C09002=1025.450,-87.514,-89.281,166.697,46.283,158.451
C09003=1025.445,-87.764,-89.270,166.694,46.286,158.451
C09004=1025.439,-88.014,-89.261,166.691,46.288,158.451
C09005=1025.433,-88.263,-89.250,166.688,46.291,158.451
C09006=1025.427,-88.513,-89.240,166.685,46.294,158.451
C09007=1025.421,-88.763,-89.230,166.683,46.297,158.452
C09008=1025.415,-89.013,-89.221,166.679,46.300,158.452
C09009=1025.409,-89.262,-89.210,166.677,46.302,158.452
C09010=1025.403,-89.512,-89.200,166.673,46.305,158.452
C09011=1025.398,-89.762,-89.190,166.670,46.308,158.452
C09012=1025.392,-90.011,-89.181,166.668,46.311,158.452
C09013=1025.387,-90.262,-89.171,166.664,46.314,158.452
C09014=1025.380,-90.511,-89.160,166.661,46.317,158.452
C09015=1025.375,-90.761,-89.150,166.659,46.319,158.453
C09016=1025.369,-91.011,-89.141,166.655,46.322,158.453
C09017=1025.363,-91.261,-89.130,166.652,46.325,158.453
C09018=1025.358,-91.510,-89.121,166.650,46.328,158.453
C09019=1025.352,-91.760,-89.111,166.646,46.331,158.453
C09020=1025.346,-92.009,-89.101,166.644,46.333,158.453
C09021=1025.340,-92.259,-89.091,166.641,46.336,158.454
C09022=1025.334,-92.509,-89.081,166.637,46.339,158.453
C09023=1025.329,-92.758,-89.071,166.635,46.341,158.454
C09024=1025.323,-93.008,-89.062,166.631,46.345,158.454
C09025=1025.317,-93.258,-89.052,166.628,46.348,158.454
C09026=1025.312,-93.508,-89.042,166.626,46.350,158.454
C09027=1025.305,-93.758,-89.032,166.622,46.353,158.454
C09028=1025.301,-94.007,-89.023,166.620,46.355,158.454
C09029=1025.294,-94.257,-89.013,166.617,46.359,158.455
C09030=1025.289,-94.507,-89.002,166.613,46.361,158.455
C09031=1025.283,-94.756,-88.993,166.611,46.364,158.455
C09032=1025.278,-95.006,-88.983,166.608,46.367,158.455
C09033=1025.272,-95.256,-88.973,166.604,46.369,158.455
C09034=1025.266,-95.506,-88.963,166.602,46.372,158.455
C09035=1025.260,-95.756,-88.954,166.598,46.375,158.455
C09036=1025.255,-96.005,-88.944,166.596,46.378,158.455
C09037=1025.249,-96.255,-88.934,166.593,46.380,158.455
C09038=1025.243,-96.505,-88.924,166.589,46.383,158.456
C09039=1025.238,-96.754,-88.915,166.587,46.386,158.456
C09040=1025.232,-97.004,-88.905,166.584,46.389,158.456
C09041=1025.226,-97.254,-88.895,166.580,46.391,158.456
C09042=1025.220,-97.504,-88.886,166.578,46.394,158.456
C09043=1025.215,-97.753,-88.876,166.575,46.397,158.456
C09044=1025.209,-98.003,-88.867,166.571,46.400,158.456
C09045=1025.203,-98.253,-88.857,166.569,46.403,158.457
C09046=1025.198,-98.502,-88.848,166.566,46.406,158.457
C09047=1025.192,-98.752,-88.838,166.562,46.408,158.457
C09048=1025.186,-99.002,-88.828,166.560,46.411,158.457
C09049=1025.181,-99.251,-88.819,166.557,46.414,158.457
C09050=1025.175,-99.502,-88.810,166.553,46.417,158.457
C09051=1025.168,-99.752,-88.801,166.551,46.420,158.457
C09052=1025.164,-100.001,-88.791,166.548,46.423,158.458
C09053=1025.157,-100.251,-88.781,166.544,46.426,158.458
C09054=1025.152,-100.501,-88.773,166.541,46.429,158.458
C09055=1025.145,-100.786,-88.761,166.538,46.432,158.458
C09056=1025.138,-101.073,-88.750,166.535,46.435,158.458
C09057=1025.132,-101.359,-88.741,166.532,46.439,158.458
C09058=1025.125,-101.644,-88.729,166.527,46.442,158.458
C09059=1025.119,-101.894,-88.720,166.525,46.445,158.459
C09060=1025.113,-102.144,-88.711,166.522,46.448,158.459
C09061=1025.108,-102.394,-88.701,166.518,46.451,158.459
C09062=1025.102,-102.644,-88.692,166.516,46.454,158.459
C09063=1025.097,-102.893,-88.683,166.512,46.456,158.459
C09064=1025.091,-103.143,-88.674,166.509,46.459,158.459
C09065=1025.085,-103.393,-88.665,166.507,46.462,158.460
C09066=1025.079,-103.642,-88.655,166.504,46.465,158.460
C09067=1025.074,-103.892,-88.645,166.500,46.468,158.460
C09068=1025.069,-104.142,-88.637,166.498,46.471,158.460
C09069=1025.062,-104.392,-88.627,166.495,46.474,158.460
C09070=1025.057,-104.641,-88.618,166.491,46.477,158.460
C09071=1025.051,-104.892,-88.609,166.488,46.480,158.460
C09072=1025.045,-105.141,-88.600,166.486,46.482,158.460
C09073=1025.040,-105.391,-88.591,166.482,46.485,158.461
C09074=1025.035,-105.640,-88.581,166.479,46.488,158.461
C09075=1025.029,-105.890,-88.572,166.477,46.491,158.461
C09076=1025.023,-106.141,-88.563,166.473,46.494,158.461
C09077=1025.017,-106.390,-88.554,166.470,46.497,158.461
C09078=1025.011,-106.640,-88.545,166.468,46.500,158.461
C09079=1025.006,-106.889,-88.536,166.465,46.503,158.462
C09080=1025.000,-107.140,-88.527,166.461,46.506,158.462
C09081=1024.994,-107.389,-88.518,166.458,46.509,158.462
C09082=1024.988,-107.639,-88.509,166.455,46.511,158.462
C09083=1024.983,-107.888,-88.500,166.452,46.514,158.462
C09084=1024.977,-108.139,-88.491,166.449,46.517,158.462
C09085=1024.971,-108.388,-88.482,166.447,46.520,158.462
C09086=1024.966,-108.638,-88.473,166.443,46.523,158.462
C09087=1024.960,-108.887,-88.463,166.440,46.526,158.463
C09088=1024.955,-109.137,-88.455,166.437,46.529,158.463
C09089=1024.949,-109.387,-88.446,166.434,46.532,158.463
C09090=1024.943,-109.637,-88.437,166.431,46.535,158.463
C09091=1024.937,-109.887,-88.428,166.428,46.538,158.463
C09092=1024.932,-110.136,-88.419,166.425,46.541,158.463
C09093=1024.926,-110.386,-88.410,166.422,46.544,158.464
C09094=1024.921,-110.636,-88.402,166.419,46.547,158.464
C09095=1024.915,-110.886,-88.392,166.416,46.550,158.464
C09096=1024.909,-111.136,-88.383,166.413,46.553,158.464
C09097=1024.904,-111.385,-88.375,166.410,46.556,158.464
C09098=1024.898,-111.635,-88.365,166.407,46.559,158.464
C09099=1024.893,-111.885,-88.357,166.404,46.562,158.464
C09100=1024.887,-112.135,-88.348,166.401,46.565,158.465
C09101=1024.880,-112.384,-88.339,166.398,46.568,158.465
C09102=1024.875,-112.634,-88.331,166.395,46.571,158.465
C09103=1024.869,-112.884,-88.322,166.391,46.574,158.465
C09104=1024.864,-113.133,-88.313,166.389,46.577,158.465
C09105=1024.858,-113.383,-88.304,166.386,46.580,158.465
C09106=1024.853,-113.633,-88.296,166.383,46.583,158.465
C09107=1024.847,-113.883,-88.287,166.380,46.586,158.466
C09108=1024.841,-114.133,-88.278,166.377,46.589,158.466
C09109=1024.836,-114.383,-88.269,166.374,46.592,158.466
C09110=1024.831,-114.632,-88.261,166.370,46.595,158.466
C09111=1024.825,-114.883,-88.252,166.368,46.598,158.466
C09112=1024.818,-115.132,-88.243,166.365,46.601,158.466
C09113=1024.813,-115.381,-88.235,166.362,46.604,158.467
C09114=1024.807,-115.632,-88.226,166.358,46.607,158.467
C09115=1024.802,-115.881,-88.217,166.356,46.610,158.467
C09116=1024.797,-116.131,-88.209,166.353,46.613,158.467
C09117=1024.791,-116.381,-88.201,166.349,46.616,158.467
C09118=1024.785,-116.631,-88.192,166.346,46.619,158.467
C09119=1024.779,-116.880,-88.183,166.344,46.622,158.467
C09120=1024.774,-117.130,-88.174,166.341,46.625,158.468
C09121=1024.768,-117.379,-88.166,166.337,46.628,158.468
C09122=1024.762,-117.628,-88.157,166.334,46.631,158.468
C09123=1024.757,-117.878,-88.149,166.332,46.634,158.468
C09124=1024.751,-118.127,-88.140,166.328,46.637,158.468
C09125=1024.746,-118.377,-88.132,166.325,46.640,158.468
C09126=1024.740,-118.626,-88.124,166.322,46.643,158.468
C09127=1024.734,-118.876,-88.115,166.320,46.646,158.469
C09128=1024.729,-119.125,-88.107,166.317,46.650,158.469
C09129=1024.724,-119.375,-88.098,166.313,46.653,158.469
///RCONF 1,0,0,0,0,0,0,0,0,0,0,0,0,0,0,0,0,0,0,0,0,0,0,0
C09130=1024.717,-119.625,-88.090,166.310,46.656,158.469
C09131=1024.712,-119.875,-88.082,166.308,46.659,158.469
C09132=1024.707,-120.125,-88.073,166.304,46.662,158.470
C09133=1024.701,-120.374,-88.065,166.301,46.665,158.470
C09134=1024.695,-120.624,-88.057,166.298,46.668,158.470
C09135=1024.690,-120.874,-88.048,166.296,46.671,158.470
C09136=1024.684,-121.124,-88.039,166.292,46.674,158.470
C09137=1024.679,-121.374,-88.031,166.289,46.677,158.470
C09138=1024.673,-121.623,-88.023,166.286,46.680,158.470
C09139=1024.667,-121.909,-88.013,166.283,46.684,158.471
C09140=1024.660,-122.196,-88.004,166.279,46.687,158.471
C09141=1024.654,-122.483,-87.995,166.276,46.691,158.471
C09142=1024.648,-122.769,-87.985,166.272,46.694,158.471
C09143=1024.642,-123.019,-87.977,166.270,46.697,158.471
C09144=1024.636,-123.268,-87.968,166.266,46.700,158.471
C09145=1024.631,-123.518,-87.960,166.263,46.703,158.471
C09146=1024.626,-123.768,-87.951,166.260,46.706,158.472
C09147=1024.619,-124.018,-87.943,166.258,46.709,158.472
C09148=1024.614,-124.268,-87.935,166.254,46.712,158.472
C09149=1024.609,-124.518,-87.927,166.251,46.716,158.472
C09150=1024.603,-124.767,-87.919,166.248,46.719,158.472
C09151=1024.598,-125.017,-87.911,166.246,46.721,158.473
C09152=1024.592,-125.266,-87.903,166.242,46.725,158.473
C09153=1024.587,-125.517,-87.895,166.239,46.728,158.473
C09154=1024.580,-125.767,-87.887,166.236,46.731,158.473
C09155=1024.575,-126.017,-87.878,166.233,46.734,158.473
C09156=1024.570,-126.266,-87.870,166.231,46.737,158.473
C09157=1024.564,-126.516,-87.862,166.227,46.740,158.474
C09158=1024.559,-126.766,-87.854,166.224,46.743,158.474
C09159=1024.553,-127.015,-87.846,166.221,46.747,158.474
C09160=1024.548,-127.265,-87.838,166.218,46.749,158.474
C09161=1024.542,-127.515,-87.830,166.215,46.752,158.474
C09162=1024.537,-127.765,-87.822,166.212,46.756,158.474
C09163=1024.531,-128.014,-87.814,166.209,46.759,158.474
C09164=1024.526,-128.264,-87.805,166.206,46.761,158.475
C09165=1024.522,-128.514,-87.796,166.203,46.764,158.474
C09166=1024.517,-128.763,-87.786,166.200,46.765,158.474
C09167=1024.515,-129.012,-87.776,166.198,46.766,158.474
C09168=1024.511,-129.262,-87.765,166.195,46.767,158.474
C09169=1024.509,-129.512,-87.754,166.193,46.767,158.474
C09170=1024.507,-129.763,-87.741,166.190,46.767,158.473
C09171=1024.506,-130.012,-87.729,166.188,46.766,158.473
C09172=1024.506,-130.262,-87.715,166.186,46.765,158.473
C09173=1024.505,-130.512,-87.702,166.183,46.763,158.472
C09174=1024.505,-130.761,-87.687,166.181,46.760,158.471
C09175=1024.506,-131.011,-87.671,166.179,46.758,158.471
C09176=1024.508,-131.261,-87.657,166.178,46.754,158.470
C09177=1024.510,-131.511,-87.640,166.176,46.751,158.469
C09178=1024.512,-131.760,-87.624,166.175,46.746,158.468
C09179=1024.515,-132.011,-87.606,166.173,46.741,158.467
C09180=1024.519,-132.260,-87.588,166.171,46.736,158.466
C09181=1024.523,-132.510,-87.570,166.169,46.730,158.465
C09182=1024.527,-132.759,-87.551,166.168,46.725,158.464
C09183=1024.230,-132.785,-87.884,166.120,47.002,158.504
C09184=1024.224,-132.536,-87.904,166.122,47.008,158.506
C09185=1024.221,-132.286,-87.923,166.123,47.014,158.507
C09186=1024.217,-132.036,-87.940,166.125,47.019,158.508
C09187=1024.215,-131.786,-87.958,166.126,47.024,158.509
C09188=1024.212,-131.537,-87.975,166.127,47.028,158.510
C09189=1024.209,-131.287,-87.991,166.130,47.032,158.511
C09190=1024.208,-131.037,-88.006,166.131,47.036,158.511
C09191=1024.207,-130.787,-88.022,166.134,47.038,158.512
C09192=1024.207,-130.537,-88.035,166.136,47.040,158.513
C09193=1024.208,-130.287,-88.049,166.137,47.042,158.513
C09194=1024.208,-130.037,-88.062,166.140,47.044,158.514
C09195=1024.209,-129.788,-88.075,166.143,47.044,158.514
C09196=1024.211,-129.539,-88.088,166.145,47.044,158.515
C09197=1024.213,-129.288,-88.100,166.147,47.044,158.515
C09198=1024.216,-129.039,-88.110,166.149,47.044,158.515
C09199=1024.220,-128.789,-88.121,166.152,47.042,158.515
C09200=1024.224,-128.539,-88.130,166.155,47.041,158.515
C09201=1024.228,-128.290,-88.140,166.158,47.039,158.515
C09202=1024.233,-128.040,-88.149,166.161,47.036,158.515
C09203=1024.238,-127.791,-88.156,166.164,47.033,158.515
C09204=1024.243,-127.541,-88.164,166.166,47.030,158.515
C09205=1024.249,-127.292,-88.172,166.170,47.027,158.515
C09206=1024.255,-127.041,-88.181,166.173,47.024,158.515
C09207=1024.260,-126.791,-88.189,166.176,47.020,158.514
C09208=1024.266,-126.541,-88.196,166.180,47.017,158.514
C09209=1024.271,-126.292,-88.205,166.182,47.014,158.514
C09210=1024.277,-126.042,-88.213,166.185,47.011,158.514
C09211=1024.282,-125.792,-88.221,166.188,47.008,158.514
C09212=1024.288,-125.543,-88.228,166.191,47.004,158.514
C09213=1024.294,-125.293,-88.237,166.195,47.001,158.514
C09214=1024.299,-125.043,-88.244,166.198,46.998,158.513
C09215=1024.305,-124.793,-88.253,166.200,46.995,158.513
C09216=1024.310,-124.543,-88.261,166.203,46.992,158.513
C09217=1024.316,-124.293,-88.269,166.206,46.988,158.513
C09218=1024.322,-124.044,-88.278,166.210,46.985,158.513
C09219=1024.327,-123.793,-88.286,166.213,46.982,158.513
C09220=1024.333,-123.544,-88.293,166.215,46.979,158.512
C09221=1024.338,-123.294,-88.302,166.218,46.976,158.512
C09222=1024.343,-123.044,-88.310,166.221,46.973,158.512
C09223=1024.349,-122.795,-88.318,166.225,46.969,158.512
C09224=1024.354,-122.545,-88.327,166.228,46.966,158.512
C09225=1024.360,-122.295,-88.336,166.230,46.963,158.512
C09226=1024.366,-122.045,-88.343,166.233,46.960,158.511
C09227=1024.371,-121.795,-88.351,166.237,46.957,158.511
C09228=1024.376,-121.545,-88.360,166.240,46.954,158.511
C09229=1024.382,-121.296,-88.368,166.242,46.951,158.511
C09230=1024.388,-121.046,-88.376,166.245,46.948,158.511
C09231=1024.394,-120.796,-88.385,166.249,46.944,158.511
C09232=1024.399,-120.546,-88.394,166.252,46.941,158.510
C09233=1024.405,-120.297,-88.401,166.255,46.938,158.510
C09234=1024.410,-120.047,-88.410,166.257,46.935,158.510
C09235=1024.415,-119.797,-88.418,166.261,46.932,158.510
C09236=1024.421,-119.547,-88.427,166.264,46.929,158.510
C09237=1024.427,-119.298,-88.435,166.267,46.926,158.510
C09238=1024.433,-119.048,-88.444,166.270,46.922,158.510
C09239=1024.438,-118.798,-88.452,166.272,46.920,158.509
C09240=1024.444,-118.548,-88.461,166.276,46.916,158.509
C09241=1024.450,-118.298,-88.469,166.279,46.913,158.509
C09242=1024.455,-118.049,-88.477,166.282,46.910,158.509
C09243=1024.460,-117.799,-88.486,166.286,46.907,158.509
C09244=1024.467,-117.513,-88.496,166.289,46.903,158.509
C09245=1024.473,-117.228,-88.505,166.292,46.900,158.508
C09246=1024.480,-116.942,-88.514,166.296,46.896,158.508
C09247=1024.486,-116.656,-88.525,166.299,46.893,158.508
C09248=1024.491,-116.407,-88.533,166.302,46.890,158.508
C09249=1024.497,-116.157,-88.541,166.305,46.887,158.508
C09250=1024.503,-115.907,-88.551,166.308,46.883,158.508
C09251=1024.509,-115.658,-88.559,166.311,46.880,158.507
C09252=1024.514,-115.408,-88.568,166.314,46.877,158.507
C09253=1024.520,-115.158,-88.577,166.317,46.874,158.507
C09254=1024.526,-114.908,-88.585,166.320,46.871,158.507
C09255=1024.531,-114.658,-88.593,166.323,46.868,158.507
C09256=1024.536,-114.409,-88.602,166.326,46.865,158.507
C09257=1024.543,-114.159,-88.611,166.330,46.862,158.507
C09258=1024.548,-113.909,-88.620,166.332,46.859,158.506
C09259=1024.554,-113.659,-88.628,166.335,46.856,158.506
C09260=1024.559,-113.409,-88.637,166.338,46.853,158.506
C09261=1024.564,-113.160,-88.646,166.342,46.850,158.506
C09262=1024.570,-112.910,-88.655,166.344,46.847,158.506
C09263=1024.576,-112.660,-88.664,166.347,46.844,158.506
C09264=1024.582,-112.410,-88.671,166.350,46.841,158.506
C09265=1024.588,-112.161,-88.681,166.354,46.838,158.505
C09266=1024.593,-111.911,-88.689,166.357,46.835,158.505
C09267=1024.598,-111.661,-88.698,166.359,46.832,158.505
C09268=1024.604,-111.411,-88.708,166.363,46.829,158.505
C09269=1024.610,-111.162,-88.716,166.366,46.825,158.505
C09270=1024.616,-110.911,-88.725,166.369,46.822,158.505
C09271=1024.621,-110.662,-88.734,166.371,46.819,158.504
C09272=1024.626,-110.412,-88.743,166.374,46.816,158.504
C09273=1024.632,-110.162,-88.751,166.378,46.813,158.504
C09274=1024.638,-109.913,-88.761,166.381,46.810,158.504
C09275=1024.644,-109.663,-88.769,166.383,46.807,158.504
C09276=1024.649,-109.413,-88.778,166.386,46.804,158.504
C09277=1024.655,-109.163,-88.787,166.390,46.801,158.503
C09278=1024.660,-108.913,-88.796,166.393,46.798,158.503
C09279=1024.666,-108.664,-88.805,166.396,46.795,158.503
C09280=1024.672,-108.420,-88.814,166.399,46.792,158.503
C09281=1024.678,-108.177,-88.822,166.402,46.789,158.503
C09282=1024.683,-107.935,-88.831,166.405,46.786,158.503
C09283=1024.689,-107.691,-88.840,166.407,46.783,158.503
C09284=1024.694,-107.447,-88.848,166.411,46.780,158.502
C09285=1024.700,-107.204,-88.858,166.414,46.777,158.502
C09286=1024.705,-106.961,-88.866,166.416,46.774,158.502
C09287=1024.711,-106.717,-88.875,166.420,46.772,158.502
C09288=1024.716,-106.468,-88.884,166.423,46.769,158.502
C09289=1024.722,-106.218,-88.893,166.425,46.766,158.502
C09290=1024.728,-105.969,-88.902,166.429,46.763,158.502
C09291=1024.733,-105.718,-88.911,166.432,46.760,158.502
C09292=1024.738,-105.469,-88.921,166.435,46.757,158.501
C09293=1024.745,-105.219,-88.930,166.437,46.754,158.501
C09294=1024.750,-104.969,-88.939,166.441,46.751,158.501
C09295=1024.756,-104.720,-88.948,166.444,46.748,158.501
C09296=1024.761,-104.470,-88.957,166.446,46.745,158.501
C09297=1024.768,-104.220,-88.966,166.449,46.742,158.501
C09298=1024.773,-103.970,-88.977,166.453,46.739,158.500
C09299=1024.778,-103.720,-88.985,166.456,46.735,158.500
C09300=1024.784,-103.470,-88.995,166.458,46.733,158.500
C09301=1024.790,-103.221,-89.003,166.462,46.730,158.500
C09302=1024.796,-102.971,-89.013,166.465,46.727,158.500
C09303=1024.801,-102.722,-89.022,166.468,46.723,158.500
C09304=1024.807,-102.471,-89.031,166.470,46.721,158.500
C09305=1024.813,-102.221,-89.041,166.474,46.718,158.499
C09306=1024.818,-101.972,-89.050,166.477,46.714,158.499
C09307=1024.824,-101.722,-89.059,166.480,46.711,158.499
C09308=1024.831,-101.423,-89.070,166.483,46.708,158.499
C09309=1024.838,-101.125,-89.082,166.486,46.705,158.499
C09310=1024.844,-100.826,-89.092,166.491,46.701,158.499
C09311=1024.851,-100.527,-89.104,166.494,46.698,158.498
C09312=1024.857,-100.277,-89.114,166.497,46.694,158.498
C09313=1024.863,-100.027,-89.122,166.500,46.691,158.498
C09314=1024.869,-99.778,-89.132,166.504,46.688,158.498
C09315=1024.874,-99.528,-89.142,166.506,46.686,158.498
C09316=1024.880,-99.278,-89.151,166.509,46.682,158.498
C09317=1024.886,-99.028,-89.160,166.512,46.679,158.498
C09318=1024.892,-98.779,-89.169,166.516,46.676,158.497
C09319=1024.898,-98.529,-89.179,166.518,46.673,158.497
C09320=1024.904,-98.280,-89.188,166.521,46.670,158.497
C09321=1024.909,-98.030,-89.198,166.525,46.667,158.497
C09322=1024.915,-97.779,-89.207,166.528,46.664,158.497
C09323=1024.920,-97.530,-89.216,166.530,46.662,158.497
C09324=1024.926,-97.280,-89.227,166.534,46.659,158.497
C09325=1024.932,-97.030,-89.236,166.537,46.656,158.496
C09326=1024.937,-96.781,-89.246,166.539,46.653,158.496
C09327=1024.943,-96.531,-89.255,166.543,46.650,158.496
C09328=1024.949,-96.281,-89.266,166.546,46.648,158.496
C09329=1024.954,-96.032,-89.275,166.548,46.645,158.496
C09330=1024.960,-95.782,-89.284,166.552,46.642,158.496
C09331=1024.966,-95.532,-89.295,166.555,46.639,158.496
C09332=1024.972,-95.282,-89.304,166.557,46.636,158.495
C09333=1024.977,-95.033,-89.314,166.561,46.634,158.495
C09334=1024.983,-94.783,-89.323,166.564,46.631,158.495
C09335=1024.988,-94.533,-89.334,166.566,46.628,158.495
C09336=1024.994,-94.283,-89.343,166.570,46.625,158.495
C09337=1024.999,-94.033,-89.353,166.573,46.622,158.495
C09338=1025.005,-93.784,-89.363,166.575,46.619,158.495
C09339=1025.011,-93.534,-89.373,166.579,46.617,158.495
C09340=1025.017,-93.284,-89.382,166.582,46.613,158.494
C09341=1025.022,-93.035,-89.393,166.584,46.611,158.494
C09342=1025.028,-92.785,-89.402,166.587,46.608,158.494
C09343=1025.034,-92.535,-89.413,166.591,46.605,158.494
C09344=1025.040,-92.285,-89.422,166.593,46.602,158.494
C09345=1025.046,-92.036,-89.431,166.597,46.599,158.494
C09346=1025.051,-91.786,-89.441,166.600,46.596,158.494
C09347=1025.057,-91.536,-89.451,166.602,46.594,158.493
C09348=1025.063,-91.286,-89.461,166.605,46.590,158.493
C09349=1025.069,-91.036,-89.471,166.609,46.587,158.493
C09350=1025.075,-90.787,-89.482,166.611,46.585,158.493
C09351=1025.080,-90.538,-89.491,166.615,46.582,158.493
C09352=1025.086,-90.288,-89.501,166.618,46.579,158.493
C09353=1025.092,-90.038,-89.511,166.620,46.576,158.493
C09354=1025.097,-89.788,-89.521,166.623,46.573,158.492
C09355=1025.104,-89.539,-89.531,166.627,46.570,158.492
C09356=1025.109,-89.288,-89.541,166.629,46.567,158.492
C09357=1025.115,-89.039,-89.550,166.632,46.565,158.492
C09358=1025.120,-88.789,-89.561,166.636,46.562,158.492
C09359=1025.126,-88.539,-89.570,166.638,46.559,158.492
C09360=1025.132,-88.290,-89.581,166.641,46.556,158.492
C09361=1025.138,-88.040,-89.591,166.645,46.553,158.491
C09362=1025.144,-87.790,-89.601,166.647,46.550,158.491
C09363=1025.150,-87.540,-89.610,166.650,46.547,158.491
C09364=1025.155,-87.291,-89.621,166.654,46.545,158.491
C09365=1025.162,-87.041,-89.631,166.657,46.542,158.491
C09366=1025.167,-86.791,-89.641,166.659,46.539,158.491
C09367=1025.173,-86.542,-89.651,166.663,46.536,158.491
C09368=1025.178,-86.292,-89.661,166.666,46.533,158.491
C09369=1025.185,-86.042,-89.671,166.668,46.530,158.490
C09370=1025.190,-85.792,-89.681,166.671,46.527,158.490
C09371=1025.196,-85.543,-89.692,166.675,46.525,158.490
C09372=1025.203,-85.259,-89.703,166.678,46.521,158.490
C09373=1025.210,-84.975,-89.714,166.681,46.518,158.490
C09374=1025.216,-84.691,-89.725,166.685,46.515,158.490
C09375=1025.223,-84.408,-89.737,166.688,46.511,158.489
C09376=1025.229,-84.158,-89.747,166.691,46.509,158.489
C09377=1025.235,-83.908,-89.758,166.694,46.506,158.489
C09378=1025.241,-83.659,-89.768,166.697,46.503,158.489
C09379=1025.246,-83.409,-89.778,166.700,46.500,158.489
C09380=1025.253,-83.159,-89.788,166.703,46.497,158.489
C09381=1025.258,-82.909,-89.798,166.707,46.494,158.489
C09382=1025.265,-82.660,-89.809,166.709,46.491,158.488
C09383=1025.270,-82.410,-89.819,166.712,46.488,158.488
C09384=1025.276,-82.160,-89.828,166.715,46.485,158.488
C09385=1025.282,-81.911,-89.839,166.718,46.482,158.488
C09386=1025.288,-81.661,-89.849,166.721,46.480,158.488
C09387=1025.294,-81.411,-89.860,166.724,46.477,158.488
C09388=1025.300,-81.162,-89.869,166.727,46.474,158.487
C09389=1025.306,-80.912,-89.880,166.730,46.471,158.487
C09390=1025.311,-80.662,-89.890,166.733,46.468,158.487
C09391=1025.318,-80.413,-89.901,166.736,46.465,158.487
C09392=1025.323,-80.163,-89.911,166.739,46.462,158.487
C09393=1025.330,-79.913,-89.921,166.742,46.459,158.487
C09394=1025.336,-79.663,-89.932,166.744,46.456,158.486
C09395=1025.341,-79.413,-89.942,166.748,46.454,158.486
C09396=1025.347,-79.164,-89.953,166.751,46.451,158.486
C09397=1025.352,-78.914,-89.963,166.754,46.448,158.486
C09398=1025.359,-78.664,-89.974,166.757,46.446,158.486
C09399=1025.365,-78.415,-89.985,166.759,46.443,158.486
C09400=1025.370,-78.165,-89.995,166.763,46.440,158.486
C09401=1025.376,-77.915,-90.006,166.766,46.437,158.486
C09402=1025.382,-77.666,-90.017,166.768,46.435,158.486
C09403=1025.388,-77.416,-90.026,166.772,46.432,158.485
C09404=1025.394,-77.166,-90.037,166.775,46.429,158.485
C09405=1025.400,-76.916,-90.048,166.777,46.426,158.485
C09406=1025.405,-76.666,-90.058,166.781,46.424,158.485
C09407=1025.411,-76.417,-90.069,166.783,46.421,158.485
C09408=1025.417,-76.167,-90.080,166.786,46.418,158.485
C09409=1025.423,-75.918,-90.090,166.790,46.415,158.484
C09410=1025.429,-75.668,-90.101,166.792,46.412,158.484
C09411=1025.435,-75.418,-90.112,166.796,46.410,158.484
C09412=1025.441,-75.168,-90.123,166.798,46.407,158.484
C09413=1025.446,-74.919,-90.134,166.801,46.404,158.484
C09414=1025.453,-74.669,-90.143,166.804,46.401,158.484
C09415=1025.458,-74.420,-90.154,166.807,46.399,158.484
C09416=1025.464,-74.170,-90.165,166.810,46.396,158.484
C09417=1025.470,-73.920,-90.176,166.813,46.393,158.483
C09418=1025.476,-73.670,-90.187,166.816,46.390,158.483
C09419=1025.481,-73.421,-90.198,166.818,46.388,158.483
C09420=1025.487,-73.170,-90.209,166.822,46.385,158.483
C09421=1025.492,-72.921,-90.220,166.825,46.382,158.483
C09422=1025.499,-72.671,-90.231,166.827,46.380,158.483
C09423=1025.504,-72.421,-90.242,166.831,46.377,158.483
C09424=1025.510,-72.172,-90.253,166.833,46.374,158.483
C09425=1025.516,-71.922,-90.263,166.837,46.372,158.483
C09426=1025.522,-71.673,-90.274,166.839,46.369,158.482
C09427=1025.528,-71.423,-90.286,166.842,46.366,158.482
C09428=1025.533,-71.173,-90.297,166.845,46.364,158.482
C09429=1025.539,-70.923,-90.308,166.848,46.361,158.482
C09430=1025.544,-70.674,-90.319,166.851,46.359,158.482
C09431=1025.550,-70.424,-90.330,166.854,46.356,158.482
C09432=1025.557,-70.174,-90.341,166.856,46.353,158.481
C09433=1025.562,-69.925,-90.352,166.860,46.351,158.481
C09434=1025.568,-69.675,-90.363,166.863,46.348,158.481
C09435=1025.574,-69.426,-90.374,166.866,46.346,158.481
C09436=1025.580,-69.144,-90.387,166.869,46.343,158.481
C09437=1025.587,-68.863,-90.399,166.872,46.340,158.481
C09438=1025.593,-68.581,-90.412,166.876,46.337,158.481
C09439=1025.600,-68.299,-90.424,166.879,46.334,158.481
C09440=1025.605,-68.050,-90.436,166.882,46.331,158.481
C09441=1025.612,-67.800,-90.447,166.885,46.329,158.480
C09442=1025.618,-67.550,-90.458,166.888,46.326,158.480
C09443=1025.623,-67.301,-90.469,166.890,46.323,158.480
C09444=1025.630,-67.051,-90.480,166.894,46.320,158.480
C09445=1025.635,-66.801,-90.491,166.896,46.318,158.480
C09446=1025.641,-66.552,-90.502,166.899,46.315,158.480
C09447=1025.647,-66.301,-90.514,166.902,46.313,158.480
///RCONF 1,0,0,1,0,0,0,0,0,0,0,0,0,0,0,0,0,0,0,0,0,0,0,0
C09448=1025.653,-66.052,-90.525,166.905,46.310,158.479
C09449=1025.658,-65.803,-90.536,166.908,46.307,158.479
C09450=1025.665,-65.553,-90.547,166.911,46.304,158.479
C09451=1025.671,-65.303,-90.558,166.914,46.301,158.479
C09452=1025.676,-65.054,-90.569,166.917,46.299,158.479
C09453=1025.683,-64.803,-90.580,166.920,46.296,158.479
C09454=1025.688,-64.554,-90.592,166.923,46.294,158.479
C09455=1025.694,-64.304,-90.604,166.926,46.291,158.479
C09456=1025.700,-64.054,-90.615,166.928,46.288,158.478
C09457=1025.706,-63.805,-90.625,166.932,46.285,158.478
C09458=1025.712,-63.555,-90.637,166.934,46.283,158.478
C09459=1025.718,-63.306,-90.648,166.937,46.280,158.478
C09460=1025.723,-63.056,-90.660,166.940,46.278,158.478
C09461=1025.729,-62.806,-90.671,166.943,46.275,158.478
C09462=1025.736,-62.557,-90.683,166.946,46.272,158.478
C09463=1025.742,-62.307,-90.694,166.949,46.269,158.477
C09464=1025.748,-62.057,-90.705,166.952,46.266,158.477
C09465=1025.754,-61.807,-90.716,166.955,46.264,158.477
C09466=1025.759,-61.558,-90.728,166.958,46.261,158.477
C09467=1025.765,-61.309,-90.739,166.960,46.258,158.477
C09468=1025.771,-61.058,-90.750,166.964,46.256,158.477
C09469=1025.777,-60.809,-90.762,166.966,46.253,158.477
C09470=1025.784,-60.559,-90.773,166.969,46.250,158.476
C09471=1025.789,-60.310,-90.784,166.972,46.248,158.476
C09472=1025.795,-60.060,-90.797,166.975,46.245,158.476
C09473=1025.801,-59.810,-90.807,166.978,46.243,158.476
C09474=1025.807,-59.560,-90.819,166.981,46.240,158.476
C09475=1025.814,-59.311,-90.830,166.984,46.237,158.476
C09476=1025.820,-59.061,-90.842,166.987,46.234,158.476
C09477=1025.825,-58.812,-90.854,166.990,46.231,158.475
C09478=1025.831,-58.562,-90.865,166.992,46.229,158.475
C09479=1025.837,-58.312,-90.876,166.996,46.226,158.475
C09480=1025.844,-58.063,-90.888,166.998,46.224,158.475
C09481=1025.850,-57.813,-90.899,167.002,46.221,158.475
C09482=1025.856,-57.563,-90.911,167.004,46.218,158.475
C09483=1025.861,-57.314,-90.922,167.007,46.215,158.475
C09484=1025.868,-57.064,-90.934,167.009,46.213,158.474
C09485=1025.874,-56.814,-90.945,167.013,46.210,158.474
C09486=1025.880,-56.565,-90.956,167.016,46.207,158.474
C09487=1025.886,-56.315,-90.969,167.019,46.205,158.474
C09488=1025.892,-56.065,-90.980,167.022,46.202,158.474
C09489=1025.898,-55.816,-90.992,167.024,46.199,158.474
C09490=1025.904,-55.566,-91.002,167.028,46.196,158.474
C09491=1025.911,-55.317,-91.014,167.030,46.194,158.473
C09492=1025.916,-55.066,-91.026,167.033,46.191,158.473
C09493=1025.922,-54.817,-91.038,167.036,46.189,158.473
C09494=1025.929,-54.567,-91.049,167.039,46.186,158.473
C09495=1025.935,-54.318,-91.061,167.041,46.183,158.473
C09496=1025.941,-54.069,-91.073,167.045,46.180,158.473
C09497=1025.947,-53.818,-91.084,167.047,46.178,158.472
C09498=1025.953,-53.569,-91.096,167.051,46.175,158.472
C09499=1025.959,-53.319,-91.107,167.054,46.172,158.472
C09500=1025.966,-53.039,-91.120,167.057,46.169,158.472
C09501=1025.973,-52.758,-91.134,167.060,46.166,158.472
C09502=1025.980,-52.478,-91.147,167.064,46.163,158.472
C09503=1025.987,-52.197,-91.160,167.066,46.160,158.471
C09504=1025.993,-51.948,-91.172,167.069,46.157,158.471
C09505=1025.999,-51.699,-91.183,167.073,46.154,158.471
C09506=1026.005,-51.448,-91.195,167.075,46.151,158.471
C09507=1026.012,-51.199,-91.207,167.078,46.148,158.471
C09508=1026.018,-50.950,-91.219,167.081,46.146,158.471
C09509=1026.024,-50.700,-91.230,167.084,46.143,158.471
C09510=1026.030,-50.450,-91.242,167.086,46.140,158.470
C09511=1026.035,-50.201,-91.255,167.090,46.138,158.470
C09512=1026.042,-49.951,-91.266,167.092,46.135,158.470
C09513=1026.048,-49.701,-91.278,167.095,46.133,158.470
C09514=1026.053,-49.451,-91.291,167.098,46.130,158.470
C09515=1026.060,-49.202,-91.302,167.101,46.128,158.470
C09516=1026.065,-48.952,-91.315,167.104,46.125,158.470
C09517=1026.071,-48.703,-91.327,167.106,46.123,158.469
C09518=1026.077,-48.453,-91.339,167.110,46.120,158.469
C09519=1026.083,-48.203,-91.351,167.112,46.118,158.469
C09520=1026.090,-47.953,-91.363,167.114,46.115,158.469
C09521=1026.095,-47.704,-91.375,167.118,46.112,158.469
C09522=1026.102,-47.454,-91.387,167.120,46.110,158.469
C09523=1026.108,-47.204,-91.400,167.124,46.107,158.469
C09524=1026.113,-46.955,-91.412,167.126,46.105,158.469
C09525=1026.119,-46.706,-91.424,167.129,46.102,158.468
C09526=1026.125,-46.456,-91.436,167.132,46.100,158.468
C09527=1026.131,-46.206,-91.449,167.135,46.097,158.468
C09528=1026.137,-45.956,-91.460,167.138,46.094,158.468
C09529=1026.143,-45.707,-91.472,167.140,46.092,158.468
C09530=1026.150,-45.457,-91.484,167.143,46.089,158.468
C09531=1026.155,-45.207,-91.497,167.146,46.087,158.468
C09532=1026.161,-44.958,-91.509,167.149,46.084,158.467
C09533=1026.167,-44.708,-91.521,167.152,46.082,158.467
C09534=1026.173,-44.458,-91.534,167.155,46.079,158.467
C09535=1026.179,-44.209,-91.546,167.157,46.076,158.467
C09536=1026.185,-43.960,-91.558,167.160,46.074,158.467
C09537=1026.191,-43.710,-91.570,167.163,46.071,158.467
C09538=1026.198,-43.460,-91.582,167.166,46.069,158.467
C09539=1026.204,-43.210,-91.595,167.169,46.066,158.466
C09540=1026.210,-42.961,-91.607,167.171,46.063,158.466
C09541=1026.216,-42.712,-91.619,167.175,46.061,158.466
C09542=1026.222,-42.462,-91.631,167.177,46.058,158.466
C09543=1026.228,-42.212,-91.644,167.180,46.056,158.466
C09544=1026.234,-41.962,-91.656,167.183,46.053,158.466
C09545=1026.240,-41.713,-91.669,167.185,46.050,158.465
C09546=1026.246,-41.463,-91.682,167.189,46.048,158.465
C09547=1026.253,-41.214,-91.694,167.191,46.045,158.465
C09548=1026.258,-40.964,-91.706,167.194,46.042,158.465
C09549=1026.264,-40.715,-91.719,167.197,46.040,158.465
C09550=1026.271,-40.465,-91.730,167.200,46.037,158.465
C09551=1026.277,-40.215,-91.743,167.203,46.035,158.465
C09552=1026.283,-39.965,-91.755,167.205,46.033,158.464
C09553=1026.289,-39.716,-91.768,167.208,46.030,158.464
C09554=1026.295,-39.466,-91.780,167.211,46.028,158.464
C09555=1026.302,-39.217,-91.793,167.214,46.025,158.464
C09556=1026.307,-38.968,-91.805,167.217,46.022,158.464
C09557=1026.313,-38.718,-91.818,167.219,46.020,158.464
C09558=1026.319,-38.468,-91.830,167.222,46.017,158.464
C09559=1026.325,-38.218,-91.843,167.225,46.015,158.463
C09560=1026.331,-37.969,-91.856,167.228,46.012,158.463
C09561=1026.337,-37.719,-91.868,167.231,46.010,158.463
C09562=1026.343,-37.469,-91.881,167.233,46.007,158.463
C09563=1026.349,-37.220,-91.894,167.237,46.005,158.463
C09564=1026.356,-36.940,-91.907,167.239,46.002,158.463
C09565=1026.363,-36.660,-91.922,167.242,45.999,158.463
C09566=1026.370,-36.380,-91.936,167.246,45.997,158.463
C09567=1026.377,-36.100,-91.951,167.249,45.994,158.462
C09568=1026.382,-35.850,-91.963,167.251,45.991,158.462
C09569=1026.389,-35.601,-91.976,167.254,45.989,158.462
C09570=1026.395,-35.351,-91.989,167.257,45.986,158.462
C09571=1026.401,-35.101,-92.002,167.260,45.984,158.462
C09572=1026.407,-34.852,-92.015,167.262,45.981,158.462
C09573=1026.413,-34.602,-92.027,167.266,45.979,158.462
C09574=1026.418,-34.353,-92.040,167.268,45.976,158.461
C09575=1026.424,-34.103,-92.053,167.271,45.974,158.461
C09576=1026.431,-33.854,-92.065,167.274,45.971,158.461
C09577=1026.437,-33.604,-92.078,167.276,45.968,158.461
C09578=1026.443,-33.355,-92.091,167.280,45.966,158.461
C09579=1026.449,-33.105,-92.103,167.282,45.963,158.461
C09580=1026.455,-32.855,-92.116,167.284,45.961,158.460
C09581=1026.461,-32.606,-92.129,167.288,45.958,158.460
C09582=1026.467,-32.356,-92.142,167.290,45.956,158.460
C09583=1026.473,-32.106,-92.155,167.293,45.953,158.460
C09584=1026.479,-31.857,-92.168,167.296,45.951,158.460
C09585=1026.485,-31.607,-92.181,167.298,45.948,158.460
C09586=1026.491,-31.358,-92.194,167.302,45.946,158.460
C09587=1026.498,-31.107,-92.207,167.304,45.943,158.459
C09588=1026.504,-30.858,-92.220,167.307,45.940,158.459
C09589=1026.510,-30.608,-92.233,167.310,45.938,158.459
C09590=1026.516,-30.359,-92.246,167.312,45.935,158.459
C09591=1026.522,-30.109,-92.258,167.315,45.933,158.459
C09592=1026.529,-29.860,-92.271,167.318,45.930,158.459
C09593=1026.535,-29.610,-92.284,167.321,45.928,158.458
C09594=1026.541,-29.361,-92.297,167.323,45.926,158.458
C09595=1026.547,-29.111,-92.310,167.326,45.923,158.458
C09596=1026.553,-28.862,-92.323,167.329,45.920,158.458
C09597=1026.559,-28.612,-92.335,167.332,45.918,158.458
C09598=1026.566,-28.363,-92.349,167.335,45.915,158.458
C09599=1026.571,-28.113,-92.361,167.337,45.913,158.458
C09600=1026.578,-27.864,-92.374,167.340,45.910,158.457
C09601=1026.584,-27.614,-92.388,167.343,45.908,158.457
C09602=1026.590,-27.364,-92.401,167.345,45.905,158.457
C09603=1026.597,-27.114,-92.414,167.349,45.903,158.457
C09604=1026.603,-26.865,-92.427,167.351,45.900,158.457
C09605=1026.608,-26.615,-92.440,167.354,45.898,158.457
C09606=1026.614,-26.366,-92.454,167.356,45.895,158.457
C09607=1026.620,-26.116,-92.467,167.359,45.893,158.457
C09608=1026.626,-25.867,-92.479,167.362,45.890,158.456
C09609=1026.632,-25.617,-92.493,167.364,45.888,158.456
C09610=1026.639,-25.367,-92.507,167.368,45.886,158.456
C09611=1026.645,-25.118,-92.520,167.370,45.883,158.456
C09612=1026.651,-24.868,-92.533,167.373,45.881,158.456
C09613=1026.657,-24.619,-92.546,167.375,45.878,158.456
C09614=1026.662,-24.369,-92.560,167.379,45.876,158.456
C09615=1026.669,-24.120,-92.573,167.381,45.873,158.455
C09616=1026.675,-23.871,-92.586,167.383,45.871,158.455
C09617=1026.681,-23.620,-92.599,167.387,45.868,158.455
C09618=1026.687,-23.370,-92.613,167.389,45.866,158.455
C09619=1026.693,-23.121,-92.626,167.391,45.863,158.455
C09620=1026.699,-22.872,-92.640,167.394,45.861,158.455
C09621=1026.705,-22.623,-92.653,167.397,45.858,158.454
C09622=1026.711,-22.372,-92.666,167.400,45.856,158.454
C09623=1026.717,-22.122,-92.680,167.402,45.854,158.454
C09624=1026.724,-21.873,-92.693,167.406,45.851,158.454
C09625=1026.730,-21.624,-92.706,167.408,45.849,158.454
C09626=1026.736,-21.375,-92.720,167.411,45.846,158.454
C09627=1026.742,-21.125,-92.733,167.413,45.844,158.454
C09628=1026.749,-20.844,-92.748,167.416,45.841,158.453
C09629=1026.756,-20.563,-92.764,167.420,45.839,158.453
C09630=1026.763,-20.282,-92.778,167.423,45.836,158.453
C09631=1026.770,-20.001,-92.794,167.425,45.833,158.453
C09632=1026.776,-19.751,-92.807,167.429,45.830,158.453
C09633=1026.782,-19.502,-92.820,167.431,45.828,158.453
C09634=1026.787,-19.253,-92.834,167.433,45.825,158.452
C09635=1026.794,-19.003,-92.847,167.436,45.823,158.452
C09636=1026.800,-18.753,-92.861,167.439,45.820,158.452
C09637=1026.806,-18.504,-92.875,167.442,45.818,158.452
C09638=1026.813,-18.254,-92.888,167.444,45.815,158.452
C09639=1026.819,-18.005,-92.902,167.448,45.813,158.452
C09640=1026.825,-17.755,-92.915,167.450,45.810,158.452
C09641=1026.831,-17.506,-92.929,167.453,45.808,158.451
C09642=1026.837,-17.256,-92.942,167.455,45.805,158.451
C09643=1026.844,-17.007,-92.956,167.458,45.803,158.451
C09644=1026.850,-16.757,-92.969,167.461,45.800,158.451
C09645=1026.856,-16.507,-92.983,167.463,45.798,158.451
///RCONF 1,0,0,0,0,0,0,0,0,0,0,0,0,0,0,0,0,0,0,0,0,0,0,0
C09646=1026.862,-16.258,-92.996,167.467,45.795,158.451
C09647=1026.868,-16.008,-93.010,167.469,45.793,158.450
C09648=1026.875,-15.758,-93.023,167.471,45.791,158.450
C09649=1026.881,-15.509,-93.037,167.474,45.788,158.450
C09650=1026.887,-15.260,-93.050,167.477,45.786,158.450
C09651=1026.893,-15.009,-93.065,167.480,45.783,158.450
C09652=1026.900,-14.761,-93.079,167.482,45.781,158.450
C09653=1026.905,-14.511,-93.092,167.484,45.778,158.449
C09654=1026.911,-14.262,-93.106,167.488,45.776,158.449
C09655=1026.917,-14.012,-93.120,167.491,45.774,158.449
C09656=1026.923,-13.762,-93.134,167.493,45.771,158.449
C09657=1026.929,-13.513,-93.147,167.495,45.769,158.449
C09658=1026.935,-13.263,-93.162,167.498,45.766,158.449
C09659=1026.942,-13.014,-93.175,167.501,45.764,158.449
C09660=1026.948,-12.764,-93.190,167.503,45.761,158.448
C09661=1026.954,-12.514,-93.203,167.506,45.759,158.448
C09662=1026.959,-12.265,-93.217,167.509,45.757,158.448
C09663=1026.966,-12.015,-93.231,167.511,45.755,158.448
C09664=1026.972,-11.766,-93.245,167.514,45.752,158.448
C09665=1026.978,-11.517,-93.258,167.517,45.750,158.448
C09666=1026.984,-11.266,-93.272,167.519,45.748,158.448
C09667=1026.991,-11.018,-93.286,167.522,45.745,158.447
C09668=1026.996,-10.768,-93.300,167.525,45.743,158.447
C09669=1027.003,-10.518,-93.314,167.527,45.740,158.447
C09670=1027.009,-10.269,-93.328,167.530,45.738,158.447
C09671=1027.015,-10.019,-93.343,167.532,45.735,158.447
C09672=1027.021,-9.770,-93.356,167.535,45.733,158.447
C09673=1027.027,-9.520,-93.370,167.538,45.730,158.447
C09674=1027.034,-9.271,-93.384,167.541,45.728,158.446
C09675=1027.039,-9.021,-93.398,167.543,45.725,158.446
C09676=1027.046,-8.771,-93.412,167.546,45.723,158.446
C09677=1027.052,-8.522,-93.426,167.549,45.720,158.446
C09678=1027.059,-8.272,-93.440,167.551,45.718,158.446
C09679=1027.064,-8.023,-93.454,167.554,45.716,158.446
C09680=1027.071,-7.773,-93.468,167.556,45.713,158.445
C09681=1027.077,-7.524,-93.482,167.559,45.711,158.445
C09682=1027.082,-7.274,-93.496,167.562,45.708,158.445
C09683=1027.089,-7.025,-93.510,167.564,45.706,158.445
C09684=1027.095,-6.775,-93.524,167.567,45.704,158.445
C09685=1027.102,-6.526,-93.538,167.569,45.701,158.445
C09686=1027.107,-6.276,-93.552,167.573,45.699,158.445
C09687=1027.114,-6.026,-93.566,167.575,45.696,158.444
C09688=1027.120,-5.777,-93.580,167.578,45.694,158.444
C09689=1027.126,-5.527,-93.595,167.580,45.691,158.444
C09690=1027.133,-5.278,-93.609,167.582,45.689,158.444
C09691=1027.139,-5.028,-93.623,167.586,45.686,158.444
C09692=1027.146,-4.746,-93.638,167.588,45.684,158.443
C09693=1027.153,-4.464,-93.655,167.591,45.681,158.443
C09694=1027.160,-4.181,-93.670,167.595,45.678,158.443
C09695=1027.167,-3.899,-93.687,167.597,45.675,158.443
C09696=1027.173,-3.649,-93.701,167.600,45.673,158.443
C09697=1027.179,-3.400,-93.715,167.602,45.671,158.443
C09698=1027.185,-3.150,-93.730,167.605,45.668,158.442
C09699=1027.191,-2.901,-93.744,167.608,45.666,158.442
C09700=1027.197,-2.651,-93.759,167.610,45.664,158.442
C09701=1027.203,-2.402,-93.773,167.613,45.661,158.442
C09702=1027.209,-2.152,-93.788,167.615,45.659,158.442
C09703=1027.215,-1.903,-93.802,167.618,45.657,158.442
C09704=1027.221,-1.653,-93.817,167.620,45.654,158.442
C09705=1027.228,-1.403,-93.832,167.623,45.652,158.441
C09706=1027.233,-1.154,-93.846,167.626,45.650,158.441
C09707=1027.239,-0.904,-93.860,167.629,45.647,158.441
C09708=1027.246,-0.655,-93.874,167.631,45.645,158.441
C09709=1027.252,-0.406,-93.889,167.634,45.643,158.441
C09710=1027.258,-0.156,-93.903,167.636,45.641,158.441
C09711=1027.264,0.094,-93.918,167.639,45.639,158.441
C09712=1027.270,0.343,-93.933,167.641,45.636,158.440
C09713=1027.276,0.593,-93.947,167.643,45.634,158.440
C09714=1027.282,0.842,-93.962,167.647,45.632,158.440
C09715=1027.288,1.092,-93.977,167.649,45.629,158.440
C09716=1027.295,1.341,-93.991,167.652,45.627,158.440
C09717=1027.300,1.591,-94.005,167.654,45.624,158.440
C09718=1027.306,1.840,-94.020,167.657,45.622,158.440
C09719=1027.312,2.089,-94.035,167.659,45.620,158.439
C09720=1027.319,2.339,-94.050,167.661,45.617,158.439
C09721=1027.325,2.589,-94.063,167.665,45.615,158.439
C09722=1027.331,2.838,-94.078,167.667,45.612,158.439
C09723=1027.338,3.088,-94.093,167.670,45.610,158.439
C09724=1027.343,3.337,-94.108,167.672,45.608,158.439
C09725=1027.350,3.586,-94.122,167.675,45.606,158.438
C09726=1027.356,3.837,-94.137,167.677,45.603,158.438
C09727=1027.362,4.085,-94.151,167.680,45.601,158.438
C09728=1027.368,4.335,-94.166,167.682,45.599,158.438
C09729=1027.374,4.585,-94.181,167.685,45.596,158.438
C09730=1027.380,4.834,-94.196,167.688,45.594,158.438
C09731=1027.387,5.083,-94.211,167.690,45.591,158.437
C09732=1027.393,5.334,-94.225,167.693,45.589,158.437
C09733=1027.398,5.583,-94.240,167.695,45.586,158.437
C09734=1027.405,5.832,-94.254,167.698,45.584,158.437
C09735=1027.411,6.082,-94.269,167.700,45.582,158.437
C09736=1027.417,6.331,-94.284,167.704,45.579,158.437
C09737=1027.423,6.581,-94.299,167.706,45.577,158.437
C09738=1027.430,6.830,-94.314,167.708,45.575,158.436
C09739=1027.436,7.079,-94.328,167.711,45.573,158.436
C09740=1027.442,7.329,-94.342,167.713,45.570,158.436
C09741=1027.449,7.579,-94.357,167.716,45.568,158.436
C09742=1027.454,7.828,-94.372,167.718,45.565,158.436
C09743=1027.461,8.077,-94.387,167.722,45.563,158.436
C09744=1027.467,8.327,-94.402,167.724,45.560,158.435
C09745=1027.474,8.577,-94.416,167.727,45.558,158.435
C09746=1027.479,8.826,-94.431,167.729,45.555,158.435
C09747=1027.486,9.075,-94.446,167.731,45.553,158.435
C09748=1027.492,9.325,-94.461,167.734,45.551,158.435
C09749=1027.499,9.575,-94.476,167.736,45.548,158.434
C09750=1027.504,9.824,-94.490,167.739,45.546,158.434
C09751=1027.511,10.073,-94.505,167.742,45.543,158.434
C09752=1027.517,10.323,-94.520,167.744,45.541,158.434
C09753=1027.523,10.573,-94.535,167.747,45.538,158.434
C09754=1027.529,10.822,-94.550,167.749,45.536,158.434
C09755=1027.536,11.071,-94.565,167.752,45.534,158.433
C09756=1027.543,11.355,-94.582,167.755,45.531,158.433
C09757=1027.550,11.640,-94.599,167.757,45.528,158.433
C09758=1027.557,11.924,-94.616,167.761,45.526,158.433
C09759=1027.565,12.209,-94.633,167.763,45.523,158.433
C09760=1027.571,12.458,-94.648,167.766,45.520,158.432
C09761=1027.578,12.708,-94.663,167.769,45.518,158.432
C09762=1027.583,12.957,-94.677,167.771,45.515,158.432
C09763=1027.590,13.206,-94.692,167.773,45.513,158.432
C09764=1027.596,13.456,-94.707,167.776,45.511,158.432
C09765=1027.603,13.706,-94.722,167.778,45.508,158.431
C09766=1027.609,13.955,-94.737,167.781,45.506,158.431
C09767=1027.615,14.205,-94.753,167.783,45.503,158.431
C09768=1027.621,14.454,-94.768,167.787,45.501,158.431
C09769=1027.627,14.703,-94.783,167.789,45.499,158.431
C09770=1027.633,14.953,-94.798,167.792,45.496,158.431
C09771=1027.639,15.203,-94.813,167.794,45.494,158.431
C09772=1027.645,15.453,-94.828,167.796,45.492,158.430
C09773=1027.652,15.701,-94.844,167.799,45.490,158.430
C09774=1027.658,15.951,-94.859,167.801,45.487,158.430
C09775=1027.664,16.201,-94.874,167.804,45.485,158.430
C09776=1027.670,16.450,-94.889,167.806,45.483,158.430
C09777=1027.677,16.699,-94.905,167.809,45.480,158.430
C09778=1027.683,16.949,-94.920,167.811,45.478,158.429
C09779=1027.688,17.198,-94.935,167.814,45.475,158.429
C09780=1027.694,17.448,-94.950,167.816,45.473,158.429
C09781=1027.701,17.697,-94.965,167.819,45.470,158.429
C09782=1027.708,17.947,-94.980,167.822,45.468,158.429
C09783=1027.713,18.197,-94.996,167.824,45.466,158.429
C09784=1027.720,18.446,-95.012,167.827,45.464,158.428
C09785=1027.726,18.695,-95.027,167.829,45.461,158.428
C09786=1027.732,18.945,-95.042,167.832,45.459,158.428
C09787=1027.738,19.194,-95.057,167.834,45.456,158.428
C09788=1027.744,19.443,-95.072,167.837,45.454,158.428
C09789=1027.751,19.693,-95.087,167.839,45.452,158.428
C09790=1027.757,19.942,-95.104,167.841,45.450,158.427
C09791=1027.763,20.192,-95.119,167.844,45.448,158.427
C09792=1027.769,20.441,-95.135,167.846,45.445,158.427
C09793=1027.775,20.691,-95.150,167.849,45.443,158.427
C09794=1027.782,20.941,-95.165,167.851,45.441,158.427
C09795=1027.788,21.190,-95.181,167.854,45.438,158.427
C09796=1027.794,21.439,-95.195,167.857,45.436,158.426
C09797=1027.800,21.688,-95.212,167.860,45.433,158.426
C09798=1027.806,21.938,-95.227,167.862,45.431,158.426
C09799=1027.812,22.187,-95.243,167.864,45.428,158.426
C09800=1027.818,22.437,-95.258,167.867,45.426,158.426
C09801=1027.825,22.686,-95.274,167.870,45.424,158.426
C09802=1027.831,22.936,-95.289,167.872,45.422,158.425
C09803=1027.837,23.185,-95.305,167.874,45.420,158.425
C09804=1027.843,23.435,-95.320,167.877,45.417,158.425
C09805=1027.850,23.684,-95.336,167.879,45.415,158.425
C09806=1027.856,23.934,-95.351,167.882,45.412,158.425
C09807=1027.862,24.183,-95.367,167.884,45.410,158.425
C09808=1027.868,24.433,-95.382,167.886,45.408,158.424
C09809=1027.874,24.682,-95.398,167.889,45.406,158.424
C09810=1027.881,24.932,-95.413,167.891,45.403,158.424
C09811=1027.887,25.181,-95.430,167.894,45.401,158.424
C09812=1027.893,25.431,-95.445,167.896,45.398,158.424
C09813=1027.900,25.680,-95.460,167.899,45.396,158.423
C09814=1027.906,25.929,-95.476,167.901,45.393,158.423
C09815=1027.912,26.179,-95.491,167.905,45.391,158.423
C09816=1027.918,26.428,-95.508,167.907,45.389,158.423
C09817=1027.924,26.678,-95.523,167.909,45.387,158.423
C09818=1027.930,26.927,-95.539,167.912,45.385,158.423
C09819=1027.937,27.176,-95.555,167.914,45.382,158.422
C09820=1027.943,27.462,-95.572,167.917,45.379,158.422
C09821=1027.950,27.748,-95.590,167.920,45.376,158.422
C09822=1027.958,28.033,-95.608,167.922,45.374,158.422
C09823=1027.965,28.319,-95.627,167.926,45.371,158.422
C09824=1027.971,28.569,-95.642,167.928,45.369,158.422
C09825=1027.978,28.818,-95.658,167.931,45.367,158.421
C09826=1027.983,29.068,-95.674,167.933,45.365,158.421
C09827=1027.989,29.317,-95.690,167.935,45.362,158.421
C09828=1027.996,29.567,-95.705,167.938,45.360,158.421
C09829=1028.002,29.816,-95.722,167.941,45.358,158.421
C09830=1028.008,30.065,-95.738,167.943,45.355,158.420
C09831=1028.014,30.314,-95.753,167.945,45.353,158.420
C09832=1028.020,30.564,-95.769,167.948,45.351,158.420
C09833=1028.026,30.814,-95.785,167.950,45.349,158.420
C09834=1028.033,31.063,-95.801,167.953,45.347,158.420
C09835=1028.039,31.312,-95.817,167.955,45.344,158.420
C09836=1028.045,31.561,-95.833,167.958,45.342,158.419
C09837=1028.051,31.811,-95.848,167.960,45.339,158.419
C09838=1028.057,32.060,-95.865,167.963,45.337,158.419
C09839=1028.063,32.310,-95.881,167.965,45.334,158.419
C09840=1028.070,32.559,-95.897,167.967,45.332,158.419
C09841=1028.076,32.808,-95.913,167.970,45.330,158.419
C09842=1028.082,33.058,-95.929,167.972,45.328,158.418
C09843=1028.088,33.308,-95.944,167.975,45.326,158.418
C09844=1028.094,33.557,-95.961,167.977,45.323,158.418
C09845=1028.100,33.806,-95.977,167.980,45.321,158.418
C09846=1028.107,34.056,-95.993,167.982,45.318,158.418
C09847=1028.113,34.305,-96.009,167.985,45.316,158.417
C09848=1028.119,34.554,-96.025,167.987,45.314,158.417
C09849=1028.126,34.803,-96.041,167.989,45.312,158.417
C09850=1028.132,35.053,-96.057,167.992,45.309,158.417
C09851=1028.138,35.303,-96.073,167.994,45.307,158.417
C09852=1028.145,35.552,-96.089,167.997,45.304,158.416
C09853=1028.150,35.802,-96.105,167.999,45.302,158.416
C09854=1028.156,36.051,-96.121,168.001,45.300,158.416
C09855=1028.162,36.300,-96.137,168.004,45.298,158.416
C09856=1028.169,36.549,-96.153,168.006,45.295,158.416
C09857=1028.175,36.799,-96.169,168.009,45.293,158.416
C09858=1028.182,37.049,-96.186,168.011,45.291,158.415
C09859=1028.188,37.298,-96.202,168.014,45.288,158.415
C09860=1028.194,37.547,-96.218,168.016,45.286,158.415
C09861=1028.200,37.797,-96.234,168.019,45.284,158.415
C09862=1028.206,38.046,-96.250,168.021,45.282,158.415
C09863=1028.212,38.295,-96.267,168.024,45.280,158.415
C09864=1028.218,38.545,-96.283,168.026,45.277,158.414
C09865=1028.225,38.795,-96.299,168.029,45.275,158.414
C09866=1028.231,39.044,-96.316,168.031,45.273,158.414
C09867=1028.237,39.293,-96.333,168.033,45.270,158.414
C09868=1028.243,39.542,-96.349,168.036,45.268,158.414
C09869=1028.249,39.791,-96.365,168.038,45.266,158.414
C09870=1028.255,40.041,-96.382,168.041,45.264,158.413
C09871=1028.261,40.291,-96.398,168.043,45.262,158.413
C09872=1028.267,40.540,-96.414,168.046,45.259,158.413
C09873=1028.274,40.789,-96.430,168.048,45.257,158.413
C09874=1028.280,41.039,-96.446,168.051,45.254,158.413
C09875=1028.286,41.288,-96.463,168.053,45.252,158.413
C09876=1028.293,41.537,-96.480,168.055,45.250,158.412
C09877=1028.299,41.787,-96.496,168.058,45.248,158.412
C09878=1028.304,42.036,-96.512,168.061,45.246,158.412
C09879=1028.310,42.285,-96.529,168.063,45.243,158.412
C09880=1028.317,42.535,-96.545,168.065,45.241,158.412
C09881=1028.323,42.785,-96.562,168.068,45.238,158.411
C09882=1028.329,43.033,-96.578,168.070,45.236,158.411
C09883=1028.335,43.283,-96.595,168.073,45.234,158.411
C09884=1028.342,43.569,-96.614,168.075,45.232,158.411
C09885=1028.349,43.854,-96.633,168.077,45.229,158.411
C09886=1028.356,44.141,-96.652,168.081,45.227,158.411
C09887=1028.363,44.426,-96.671,168.083,45.224,158.410
C09888=1028.369,44.675,-96.687,168.086,45.222,158.410
C09889=1028.375,44.925,-96.705,168.089,45.220,158.410
C09890=1028.381,45.174,-96.722,168.091,45.217,158.410
C09891=1028.387,45.424,-96.738,168.093,45.215,158.410
C09892=1028.393,45.672,-96.755,168.096,45.213,158.410
C09893=1028.399,45.922,-96.771,168.098,45.211,158.409
C09894=1028.405,46.172,-96.788,168.100,45.209,158.409
C09895=1028.411,46.421,-96.805,168.102,45.207,158.409
C09896=1028.417,46.670,-96.822,168.105,45.204,158.409
C09897=1028.424,46.919,-96.839,168.107,45.202,158.409
C09898=1028.430,47.169,-96.855,168.110,45.200,158.409
C09899=1028.435,47.418,-96.872,168.112,45.198,158.408
C09900=1028.441,47.667,-96.889,168.115,45.196,158.408
C09901=1028.448,47.917,-96.906,168.117,45.194,158.408
C09902=1028.454,48.166,-96.923,168.119,45.191,158.408
C09903=1028.460,48.415,-96.939,168.122,45.189,158.408
C09904=1028.466,48.666,-96.956,168.125,45.187,158.408
C09905=1028.472,48.914,-96.973,168.127,45.184,158.407
C09906=1028.478,49.164,-96.989,168.129,45.182,158.407
C09907=1028.485,49.413,-97.007,168.132,45.180,158.407
C09908=1028.490,49.663,-97.023,168.134,45.178,158.407
C09909=1028.496,49.912,-97.040,168.137,45.176,158.407
C09910=1028.502,50.161,-97.057,168.139,45.174,158.407
C09911=1028.509,50.410,-97.074,168.142,45.171,158.406
C09912=1028.515,50.660,-97.090,168.143,45.169,158.406
C09913=1028.521,50.909,-97.108,168.146,45.166,158.406
C09914=1028.527,51.159,-97.124,168.148,45.164,158.406
C09915=1028.533,51.408,-97.141,168.151,45.162,158.406
C09916=1028.540,51.658,-97.158,168.153,45.160,158.405
C09917=1028.545,51.907,-97.176,168.156,45.158,158.405
C09918=1028.551,52.156,-97.192,168.158,45.155,158.405
C09919=1028.558,52.405,-97.209,168.160,45.153,158.405
C09920=1028.564,52.655,-97.225,168.163,45.151,158.405
C09921=1028.570,52.904,-97.243,168.165,45.149,158.404
C09922=1028.576,53.154,-97.260,168.168,45.147,158.404
C09923=1028.582,53.403,-97.277,168.170,45.144,158.404
C09924=1028.588,53.652,-97.293,168.173,45.142,158.404
C09925=1028.595,53.901,-97.310,168.175,45.139,158.404
C09926=1028.601,54.150,-97.328,168.178,45.137,158.404
C09927=1028.607,54.400,-97.344,168.180,45.135,158.403
C09928=1028.614,54.649,-97.361,168.183,45.133,158.403
C09929=1028.620,54.899,-97.378,168.185,45.131,158.403
C09930=1028.626,55.148,-97.396,168.187,45.128,158.403
C09931=1028.632,55.397,-97.413,168.190,45.126,158.403
C09932=1028.639,55.647,-97.429,168.192,45.123,158.402
C09933=1028.645,55.896,-97.446,168.195,45.121,158.402
C09934=1028.651,56.146,-97.463,168.197,45.119,158.402
C09935=1028.657,56.395,-97.480,168.200,45.117,158.402
C09936=1028.663,56.644,-97.497,168.202,45.114,158.402
C09937=1028.670,56.894,-97.514,168.205,45.112,158.402
C09938=1028.675,57.143,-97.532,168.207,45.110,158.401
C09939=1028.682,57.392,-97.549,168.209,45.107,158.401
C09940=1028.688,57.641,-97.565,168.212,45.105,158.401
C09941=1028.694,57.891,-97.583,168.214,45.103,158.401
C09942=1028.700,58.140,-97.600,168.217,45.101,158.401
C09943=1028.707,58.390,-97.617,168.218,45.098,158.400
C09944=1028.713,58.639,-97.634,168.221,45.096,158.400
C09945=1028.719,58.888,-97.652,168.223,45.094,158.400
C09946=1028.725,59.138,-97.668,168.226,45.092,158.400
C09947=1028.732,59.387,-97.685,168.228,45.089,158.400
C09948=1028.738,59.672,-97.705,168.231,45.086,158.399
C09949=1028.746,59.957,-97.725,168.234,45.083,158.399
C09950=1028.754,60.243,-97.744,168.237,45.081,158.399
C09951=1028.761,60.528,-97.764,168.239,45.078,158.399
C09952=1028.767,60.778,-97.781,168.242,45.076,158.398
C09953=1028.773,61.027,-97.797,168.244,45.073,158.398
C09954=1028.779,61.277,-97.815,168.247,45.071,158.398
C09955=1028.786,61.526,-97.832,168.249,45.069,158.398
C09956=1028.793,61.775,-97.850,168.252,45.067,158.398
C09957=1028.798,62.025,-97.866,168.254,45.064,158.397
C09958=1028.805,62.274,-97.884,168.256,45.062,158.397
C09959=1028.811,62.523,-97.901,168.259,45.059,158.397
C09960=1028.818,62.772,-97.918,168.261,45.057,158.397
C09961=1028.824,63.022,-97.936,168.264,45.055,158.397
C09962=1028.830,63.271,-97.953,168.266,45.052,158.396
C09963=1028.837,63.521,-97.970,168.269,45.050,158.396
C09964=1028.842,63.770,-97.987,168.271,45.048,158.396
C09965=1028.848,64.020,-98.005,168.273,45.045,158.396
C09966=1028.855,64.268,-98.022,168.276,45.043,158.396
C09967=1028.861,64.518,-98.040,168.278,45.041,158.395
C09968=1028.867,64.767,-98.057,168.281,45.039,158.395
C09969=1028.873,65.016,-98.075,168.283,45.037,158.395
C09970=1028.879,65.265,-98.092,168.286,45.034,158.395
C09971=1028.885,65.515,-98.110,168.288,45.032,158.395
C09972=1028.892,65.764,-98.127,168.291,45.030,158.395
C09973=1028.898,66.013,-98.145,168.293,45.028,158.394
C09974=1028.904,66.263,-98.163,168.295,45.025,158.394
C09975=1028.910,66.512,-98.180,168.297,45.023,158.394
C09976=1028.916,66.762,-98.198,168.300,45.021,158.394
C09977=1028.923,67.010,-98.215,168.302,45.019,158.394
C09978=1028.929,67.260,-98.232,168.304,45.017,158.393
C09979=1028.935,67.510,-98.250,168.307,45.014,158.393
C09980=1028.941,67.759,-98.267,168.309,45.012,158.393
C09981=1028.947,68.008,-98.285,168.312,45.010,158.393
C09982=1028.953,68.257,-98.303,168.314,45.007,158.393
C09983=1028.960,68.507,-98.320,168.317,45.005,158.393
C09984=1028.967,68.830,-98.343,168.320,45.002,158.392
C09985=1028.975,69.153,-98.366,168.323,45.000,158.392
C09986=1028.984,69.476,-98.390,168.326,44.997,158.392
C09987=1028.991,69.799,-98.413,168.329,44.993,158.392
C09988=1028.997,70.048,-98.430,168.331,44.991,158.391
C09989=1029.004,70.298,-98.448,168.334,44.989,158.391
C09990=1029.010,70.548,-98.466,168.336,44.987,158.391
C09991=1029.015,70.797,-98.483,168.339,44.985,158.391
C09992=1029.022,71.046,-98.501,168.341,44.983,158.391
C09993=1029.028,71.295,-98.519,168.344,44.980,158.390
C09994=1029.034,71.544,-98.537,168.346,44.978,158.390
C09995=1029.040,71.794,-98.555,168.349,44.976,158.390
C09996=1029.046,72.043,-98.572,168.351,44.974,158.390
//INST
///DATE 2021/06/17 10:58
///ATTR SC,RW,RJ
////FRAME ROBOT
///GROUP1 RB1
NOP
MOVL C00000 V=800.0 PL=0
MOVL C00001 V=800.0 PL=0
MOVL C00002 V=800.0 PL=0
MOVL C00003 V=800.0 PL=0
MOVL C00004 V=800.0 PL=0
MOVL C00005 V=800.0 PL=0
MOVL C00006 V=800.0 PL=0
MOVL C00007 V=800.0 PL=0
MOVL C00008 V=800.0 PL=0
MOVL C00009 V=800.0 PL=0
MOVL C00010 V=800.0 PL=0
MOVL C00011 V=800.0 PL=0
MOVL C00012 V=800.0 PL=0
MOVL C00013 V=800.0 PL=0
MOVL C00014 V=800.0 PL=0
MOVL C00015 V=800.0 PL=0
MOVL C00016 V=800.0 PL=0
MOVL C00017 V=800.0 PL=0
MOVL C00018 V=800.0 PL=0
MOVL C00019 V=800.0 PL=0
MOVL C00020 V=800.0 PL=0
MOVL C00021 V=800.0 PL=0
MOVL C00022 V=800.0 PL=0
MOVL C00023 V=800.0 PL=0
MOVL C00024 V=800.0 PL=0
MOVL C00025 V=800.0 PL=0
MOVL C00026 V=800.0 PL=0
MOVL C00027 V=800.0 PL=0
MOVL C00028 V=800.0 PL=0
MOVL C00029 V=800.0 PL=0
MOVL C00030 V=800.0 PL=0
MOVL C00031 V=800.0 PL=0
MOVL C00032 V=800.0 PL=0
MOVL C00033 V=800.0 PL=0
MOVL C00034 V=800.0 PL=0
MOVL C00035 V=800.0 PL=0
MOVL C00036 V=800.0 PL=0
MOVL C00037 V=800.0 PL=0
MOVL C00038 V=800.0 PL=0
MOVL C00039 V=800.0 PL=0
MOVL C00040 V=800.0 PL=0
MOVL C00041 V=800.0 PL=0
MOVL C00042 V=800.0 PL=0
MOVL C00043 V=800.0 PL=0
MOVL C00044 V=800.0 PL=0
MOVL C00045 V=800.0 PL=0
MOVL C00046 V=800.0 PL=0
MOVL C00047 V=800.0 PL=0
MOVL C00048 V=800.0 PL=0
MOVL C00049 V=800.0 PL=0
MOVL C00050 V=800.0 PL=0
MOVL C00051 V=800.0 PL=0
MOVL C00052 V=800.0 PL=0
MOVL C00053 V=800.0 PL=0
MOVL C00054 V=800.0 PL=0
MOVL C00055 V=800.0 PL=0
MOVL C00056 V=800.0 PL=0
MOVL C00057 V=800.0 PL=0
MOVL C00058 V=800.0 PL=0
MOVL C00059 V=800.0 PL=0
MOVL C00060 V=800.0 PL=0
MOVL C00061 V=800.0 PL=0
MOVL C00062 V=800.0 PL=0
MOVL C00063 V=800.0 PL=0
MOVL C00064 V=800.0 PL=0
MOVL C00065 V=800.0 PL=0
MOVL C00066 V=800.0 PL=0
MOVL C00067 V=800.0 PL=0
MOVL C00068 V=800.0 PL=0
MOVL C00069 V=800.0 PL=0
MOVL C00070 V=800.0 PL=0
MOVL C00071 V=800.0 PL=0
MOVL C00072 V=800.0 PL=0
MOVL C00073 V=800.0 PL=0
MOVL C00074 V=800.0 PL=0
MOVL C00075 V=800.0 PL=0
MOVL C00076 V=800.0 PL=0
MOVL C00077 V=800.0 PL=0
MOVL C00078 V=800.0 PL=0
MOVL C00079 V=800.0 PL=0
MOVL C00080 V=800.0 PL=0
MOVL C00081 V=800.0 PL=0
MOVL C00082 V=800.0 PL=0
MOVL C00083 V=800.0 PL=0
MOVL C00084 V=800.0 PL=0
MOVL C00085 V=800.0 PL=0
MOVL C00086 V=800.0 PL=0
MOVL C00087 V=800.0 PL=0
MOVL C00088 V=800.0 PL=0
MOVL C00089 V=800.0 PL=0
MOVL C00090 V=800.0 PL=0
MOVL C00091 V=800.0 PL=0
MOVL C00092 V=800.0 PL=0
MOVL C00093 V=800.0 PL=0
MOVL C00094 V=800.0 PL=0
MOVL C00095 V=800.0 PL=0
MOVL C00096 V=800.0 PL=0
MOVL C00097 V=800.0 PL=0
MOVL C00098 V=800.0 PL=0
MOVL C00099 V=800.0 PL=0
MOVL C00100 V=800.0 PL=0
MOVL C00101 V=800.0 PL=0
MOVL C00102 V=800.0 PL=0
MOVL C00103 V=800.0 PL=0
MOVL C00104 V=800.0 PL=0
MOVL C00105 V=800.0 PL=0
MOVL C00106 V=800.0 PL=0
MOVL C00107 V=800.0 PL=0
MOVL C00108 V=800.0 PL=0
MOVL C00109 V=800.0 PL=0
MOVL C00110 V=800.0 PL=0
MOVL C00111 V=800.0 PL=0
MOVL C00112 V=800.0 PL=0
MOVL C00113 V=800.0 PL=0
MOVL C00114 V=800.0 PL=0
MOVL C00115 V=800.0 PL=0
MOVL C00116 V=800.0 PL=0
MOVL C00117 V=800.0 PL=0
MOVL C00118 V=800.0 PL=0
MOVL C00119 V=800.0 PL=0
MOVL C00120 V=800.0 PL=0
MOVL C00121 V=800.0 PL=0
MOVL C00122 V=800.0 PL=0
MOVL C00123 V=800.0 PL=0
MOVL C00124 V=800.0 PL=0
MOVL C00125 V=800.0 PL=0
MOVL C00126 V=800.0 PL=0
MOVL C00127 V=800.0 PL=0
MOVL C00128 V=800.0 PL=0
MOVL C00129 V=800.0 PL=0
MOVL C00130 V=800.0 PL=0
MOVL C00131 V=800.0 PL=0
MOVL C00132 V=800.0 PL=0
MOVL C00133 V=800.0 PL=0
MOVL C00134 V=800.0 PL=0
MOVL C00135 V=800.0 PL=0
MOVL C00136 V=800.0 PL=0
MOVL C00137 V=800.0 PL=0
MOVL C00138 V=800.0 PL=0
MOVL C00139 V=800.0 PL=0
MOVL C00140 V=800.0 PL=0
MOVL C00141 V=800.0 PL=0
MOVL C00142 V=800.0 PL=0
MOVL C00143 V=800.0 PL=0
MOVL C00144 V=800.0 PL=0
MOVL C00145 V=800.0 PL=0
MOVL C00146 V=800.0 PL=0
MOVL C00147 V=800.0 PL=0
MOVL C00148 V=800.0 PL=0
MOVL C00149 V=800.0 PL=0
MOVL C00150 V=800.0 PL=0
MOVL C00151 V=800.0 PL=0
MOVL C00152 V=800.0 PL=0
MOVL C00153 V=800.0 PL=0
MOVL C00154 V=800.0 PL=0
MOVL C00155 V=800.0 PL=0
MOVL C00156 V=800.0 PL=0
MOVL C00157 V=800.0 PL=0
MOVL C00158 V=800.0 PL=0
MOVL C00159 V=800.0 PL=0
MOVL C00160 V=800.0 PL=0
MOVL C00161 V=800.0 PL=0
MOVL C00162 V=800.0 PL=0
MOVL C00163 V=800.0 PL=0
MOVL C00164 V=800.0 PL=0
MOVL C00165 V=800.0 PL=0
MOVL C00166 V=800.0 PL=0
MOVL C00167 V=800.0 PL=0
MOVL C00168 V=800.0 PL=0
MOVL C00169 V=800.0 PL=0
MOVL C00170 V=800.0 PL=0
MOVL C00171 V=800.0 PL=0
MOVL C00172 V=800.0 PL=0
MOVL C00173 V=800.0 PL=0
MOVL C00174 V=800.0 PL=0
MOVL C00175 V=800.0 PL=0
MOVL C00176 V=800.0 PL=0
MOVL C00177 V=800.0 PL=0
MOVL C00178 V=800.0 PL=0
MOVL C00179 V=800.0 PL=0
MOVL C00180 V=800.0 PL=0
MOVL C00181 V=800.0 PL=0
MOVL C00182 V=800.0 PL=0
MOVL C00183 V=800.0 PL=0
MOVL C00184 V=800.0 PL=0
MOVL C00185 V=800.0 PL=0
MOVL C00186 V=800.0 PL=0
MOVL C00187 V=800.0 PL=0
MOVL C00188 V=800.0 PL=0
MOVL C00189 V=800.0 PL=0
MOVL C00190 V=800.0 PL=0
MOVL C00191 V=800.0 PL=0
MOVL C00192 V=800.0 PL=0
MOVL C00193 V=800.0 PL=0
MOVL C00194 V=800.0 PL=0
MOVL C00195 V=800.0 PL=0
MOVL C00196 V=800.0 PL=0
MOVL C00197 V=800.0 PL=0
MOVL C00198 V=800.0 PL=0
MOVL C00199 V=800.0 PL=0
MOVL C00200 V=800.0 PL=0
MOVL C00201 V=800.0 PL=0
MOVL C00202 V=800.0 PL=0
MOVL C00203 V=800.0 PL=0
MOVL C00204 V=800.0 PL=0
MOVL C00205 V=800.0 PL=0
MOVL C00206 V=800.0 PL=0
MOVL C00207 V=800.0 PL=0
MOVL C00208 V=800.0 PL=0
MOVL C00209 V=800.0 PL=0
MOVL C00210 V=800.0 PL=0
MOVL C00211 V=800.0 PL=0
MOVL C00212 V=800.0 PL=0
MOVL C00213 V=800.0 PL=0
MOVL C00214 V=800.0 PL=0
MOVL C00215 V=800.0 PL=0
MOVL C00216 V=800.0 PL=0
MOVL C00217 V=800.0 PL=0
MOVL C00218 V=800.0 PL=0
MOVL C00219 V=800.0 PL=0
MOVL C00220 V=800.0 PL=0
MOVL C00221 V=800.0 PL=0
MOVL C00222 V=800.0 PL=0
MOVL C00223 V=800.0 PL=0
MOVL C00224 V=800.0 PL=0
MOVL C00225 V=800.0 PL=0
MOVL C00226 V=800.0 PL=0
MOVL C00227 V=800.0 PL=0
MOVL C00228 V=800.0 PL=0
MOVL C00229 V=800.0 PL=0
MOVL C00230 V=800.0 PL=0
MOVL C00231 V=800.0 PL=0
MOVL C00232 V=800.0 PL=0
MOVL C00233 V=800.0 PL=0
MOVL C00234 V=800.0 PL=0
MOVL C00235 V=800.0 PL=0
MOVL C00236 V=800.0 PL=0
MOVL C00237 V=800.0 PL=0
MOVL C00238 V=800.0 PL=0
MOVL C00239 V=800.0 PL=0
MOVL C00240 V=800.0 PL=0
MOVL C00241 V=800.0 PL=0
MOVL C00242 V=800.0 PL=0
MOVL C00243 V=800.0 PL=0
MOVL C00244 V=800.0 PL=0
MOVL C00245 V=800.0 PL=0
MOVL C00246 V=800.0 PL=0
MOVL C00247 V=800.0 PL=0
MOVL C00248 V=800.0 PL=0
MOVL C00249 V=800.0 PL=0
MOVL C00250 V=800.0 PL=0
MOVL C00251 V=800.0 PL=0
MOVL C00252 V=800.0 PL=0
MOVL C00253 V=800.0 PL=0
MOVL C00254 V=800.0 PL=0
MOVL C00255 V=800.0 PL=0
MOVL C00256 V=800.0 PL=0
MOVL C00257 V=800.0 PL=0
MOVL C00258 V=800.0 PL=0
MOVL C00259 V=800.0 PL=0
MOVL C00260 V=800.0 PL=0
MOVL C00261 V=800.0 PL=0
MOVL C00262 V=800.0 PL=0
MOVL C00263 V=800.0 PL=0
MOVL C00264 V=800.0 PL=0
MOVL C00265 V=800.0 PL=0
MOVL C00266 V=800.0 PL=0
MOVL C00267 V=800.0 PL=0
MOVL C00268 V=800.0 PL=0
MOVL C00269 V=800.0 PL=0
MOVL C00270 V=800.0 PL=0
MOVL C00271 V=800.0 PL=0
MOVL C00272 V=800.0 PL=0
MOVL C00273 V=800.0 PL=0
MOVL C00274 V=800.0 PL=0
MOVL C00275 V=800.0 PL=0
MOVL C00276 V=800.0 PL=0
MOVL C00277 V=800.0 PL=0
MOVL C00278 V=800.0 PL=0
MOVL C00279 V=800.0 PL=0
MOVL C00280 V=800.0 PL=0
MOVL C00281 V=800.0 PL=0
MOVL C00282 V=800.0 PL=0
MOVL C00283 V=800.0 PL=0
MOVL C00284 V=800.0 PL=0
MOVL C00285 V=800.0 PL=0
MOVL C00286 V=800.0 PL=0
MOVL C00287 V=800.0 PL=0
MOVL C00288 V=800.0 PL=0
MOVL C00289 V=800.0 PL=0
MOVL C00290 V=800.0 PL=0
MOVL C00291 V=800.0 PL=0
MOVL C00292 V=800.0 PL=0
MOVL C00293 V=800.0 PL=0
MOVL C00294 V=800.0 PL=0
MOVL C00295 V=800.0 PL=0
MOVL C00296 V=800.0 PL=0
MOVL C00297 V=800.0 PL=0
MOVL C00298 V=800.0 PL=0
MOVL C00299 V=800.0 PL=0
MOVL C00300 V=800.0 PL=0
MOVL C00301 V=800.0 PL=0
MOVL C00302 V=800.0 PL=0
MOVL C00303 V=800.0 PL=0
MOVL C00304 V=800.0 PL=0
MOVL C00305 V=800.0 PL=0
MOVL C00306 V=800.0 PL=0
MOVL C00307 V=800.0 PL=0
MOVL C00308 V=800.0 PL=0
MOVL C00309 V=800.0 PL=0
MOVL C00310 V=800.0 PL=0
MOVL C00311 V=800.0 PL=0
MOVL C00312 V=800.0 PL=0
MOVL C00313 V=800.0 PL=0
MOVL C00314 V=800.0 PL=0
MOVL C00315 V=800.0 PL=0
MOVL C00316 V=800.0 PL=0
MOVL C00317 V=800.0 PL=0
MOVL C00318 V=800.0 PL=0
MOVL C00319 V=800.0 PL=0
MOVL C00320 V=800.0 PL=0
MOVL C00321 V=800.0 PL=0
MOVL C00322 V=800.0 PL=0
MOVL C00323 V=800.0 PL=0
MOVL C00324 V=800.0 PL=0
MOVL C00325 V=800.0 PL=0
MOVL C00326 V=800.0 PL=0
MOVL C00327 V=800.0 PL=0
MOVL C00328 V=800.0 PL=0
MOVL C00329 V=800.0 PL=0
MOVL C00330 V=800.0 PL=0
MOVL C00331 V=800.0 PL=0
MOVL C00332 V=800.0 PL=0
MOVL C00333 V=800.0 PL=0
MOVL C00334 V=800.0 PL=0
MOVL C00335 V=800.0 PL=0
MOVL C00336 V=800.0 PL=0
MOVL C00337 V=800.0 PL=0
MOVL C00338 V=800.0 PL=0
MOVL C00339 V=800.0 PL=0
MOVL C00340 V=800.0 PL=0
MOVL C00341 V=800.0 PL=0
MOVL C00342 V=800.0 PL=0
MOVL C00343 V=800.0 PL=0
MOVL C00344 V=800.0 PL=0
MOVL C00345 V=800.0 PL=0
MOVL C00346 V=800.0 PL=0
MOVL C00347 V=800.0 PL=0
MOVL C00348 V=800.0 PL=0
MOVL C00349 V=800.0 PL=0
MOVL C00350 V=800.0 PL=0
MOVL C00351 V=800.0 PL=0
MOVL C00352 V=800.0 PL=0
MOVL C00353 V=800.0 PL=0
MOVL C00354 V=800.0 PL=0
MOVL C00355 V=800.0 PL=0
MOVL C00356 V=800.0 PL=0
MOVL C00357 V=800.0 PL=0
MOVL C00358 V=800.0 PL=0
MOVL C00359 V=800.0 PL=0
MOVL C00360 V=800.0 PL=0
MOVL C00361 V=800.0 PL=0
MOVL C00362 V=800.0 PL=0
MOVL C00363 V=800.0 PL=0
MOVL C00364 V=800.0 PL=0
MOVL C00365 V=800.0 PL=0
MOVL C00366 V=800.0 PL=0
MOVL C00367 V=800.0 PL=0
MOVL C00368 V=800.0 PL=0
MOVL C00369 V=800.0 PL=0
MOVL C00370 V=800.0 PL=0
MOVL C00371 V=800.0 PL=0
MOVL C00372 V=800.0 PL=0
MOVL C00373 V=800.0 PL=0
MOVL C00374 V=800.0 PL=0
MOVL C00375 V=800.0 PL=0
MOVL C00376 V=800.0 PL=0
MOVL C00377 V=800.0 PL=0
MOVL C00378 V=800.0 PL=0
MOVL C00379 V=800.0 PL=0
MOVL C00380 V=800.0 PL=0
MOVL C00381 V=800.0 PL=0
MOVL C00382 V=800.0 PL=0
MOVL C00383 V=800.0 PL=0
MOVL C00384 V=800.0 PL=0
MOVL C00385 V=800.0 PL=0
MOVL C00386 V=800.0 PL=0
MOVL C00387 V=800.0 PL=0
MOVL C00388 V=800.0 PL=0
MOVL C00389 V=800.0 PL=0
MOVL C00390 V=800.0 PL=0
MOVL C00391 V=800.0 PL=0
MOVL C00392 V=800.0 PL=0
MOVL C00393 V=800.0 PL=0
MOVL C00394 V=800.0 PL=0
MOVL C00395 V=800.0 PL=0
MOVL C00396 V=800.0 PL=0
MOVL C00397 V=800.0 PL=0
MOVL C00398 V=800.0 PL=0
MOVL C00399 V=800.0 PL=0
MOVL C00400 V=800.0 PL=0
MOVL C00401 V=800.0 PL=0
MOVL C00402 V=800.0 PL=0
MOVL C00403 V=800.0 PL=0
MOVL C00404 V=800.0 PL=0
MOVL C00405 V=800.0 PL=0
MOVL C00406 V=800.0 PL=0
MOVL C00407 V=800.0 PL=0
MOVL C00408 V=800.0 PL=0
MOVL C00409 V=800.0 PL=0
MOVL C00410 V=800.0 PL=0
MOVL C00411 V=800.0 PL=0
MOVL C00412 V=800.0 PL=0
MOVL C00413 V=800.0 PL=0
MOVL C00414 V=800.0 PL=0
MOVL C00415 V=800.0 PL=0
MOVL C00416 V=800.0 PL=0
MOVL C00417 V=800.0 PL=0
MOVL C00418 V=800.0 PL=0
MOVL C00419 V=800.0 PL=0
MOVL C00420 V=800.0 PL=0
MOVL C00421 V=800.0 PL=0
MOVL C00422 V=800.0 PL=0
MOVL C00423 V=800.0 PL=0
MOVL C00424 V=800.0 PL=0
MOVL C00425 V=800.0 PL=0
MOVL C00426 V=800.0 PL=0
MOVL C00427 V=800.0 PL=0
MOVL C00428 V=800.0 PL=0
MOVL C00429 V=800.0 PL=0
MOVL C00430 V=800.0 PL=0
MOVL C00431 V=800.0 PL=0
MOVL C00432 V=800.0 PL=0
MOVL C00433 V=800.0 PL=0
MOVL C00434 V=800.0 PL=0
MOVL C00435 V=800.0 PL=0
MOVL C00436 V=800.0 PL=0
MOVL C00437 V=800.0 PL=0
MOVL C00438 V=800.0 PL=0
MOVL C00439 V=800.0 PL=0
MOVL C00440 V=800.0 PL=0
MOVL C00441 V=800.0 PL=0
MOVL C00442 V=800.0 PL=0
MOVL C00443 V=800.0 PL=0
MOVL C00444 V=800.0 PL=0
MOVL C00445 V=800.0 PL=0
MOVL C00446 V=800.0 PL=0
MOVL C00447 V=800.0 PL=0
MOVL C00448 V=800.0 PL=0
MOVL C00449 V=800.0 PL=0
MOVL C00450 V=800.0 PL=0
MOVL C00451 V=800.0 PL=0
MOVL C00452 V=800.0 PL=0
MOVL C00453 V=800.0 PL=0
MOVL C00454 V=800.0 PL=0
MOVL C00455 V=800.0 PL=0
MOVL C00456 V=800.0 PL=0
MOVL C00457 V=800.0 PL=0
MOVL C00458 V=800.0 PL=0
MOVL C00459 V=800.0 PL=0
MOVL C00460 V=800.0 PL=0
MOVL C00461 V=800.0 PL=0
MOVL C00462 V=800.0 PL=0
MOVL C00463 V=800.0 PL=0
MOVL C00464 V=800.0 PL=0
MOVL C00465 V=800.0 PL=0
MOVL C00466 V=800.0 PL=0
MOVL C00467 V=800.0 PL=0
MOVL C00468 V=800.0 PL=0
MOVL C00469 V=800.0 PL=0
MOVL C00470 V=800.0 PL=0
MOVL C00471 V=800.0 PL=0
MOVL C00472 V=800.0 PL=0
MOVL C00473 V=800.0 PL=0
MOVL C00474 V=800.0 PL=0
MOVL C00475 V=800.0 PL=0
MOVL C00476 V=800.0 PL=0
MOVL C00477 V=800.0 PL=0
MOVL C00478 V=800.0 PL=0
MOVL C00479 V=800.0 PL=0
MOVL C00480 V=800.0 PL=0
MOVL C00481 V=800.0 PL=0
MOVL C00482 V=800.0 PL=0
MOVL C00483 V=800.0 PL=0
MOVL C00484 V=800.0 PL=0
MOVL C00485 V=800.0 PL=0
MOVL C00486 V=800.0 PL=0
MOVL C00487 V=800.0 PL=0
MOVL C00488 V=800.0 PL=0
MOVL C00489 V=800.0 PL=0
MOVL C00490 V=800.0 PL=0
MOVL C00491 V=800.0 PL=0
MOVL C00492 V=800.0 PL=0
MOVL C00493 V=800.0 PL=0
MOVL C00494 V=800.0 PL=0
MOVL C00495 V=800.0 PL=0
MOVL C00496 V=800.0 PL=0
MOVL C00497 V=800.0 PL=0
MOVL C00498 V=800.0 PL=0
MOVL C00499 V=800.0 PL=0
MOVL C00500 V=800.0 PL=0
MOVL C00501 V=800.0 PL=0
MOVL C00502 V=800.0 PL=0
MOVL C00503 V=800.0 PL=0
MOVL C00504 V=800.0 PL=0
MOVL C00505 V=800.0 PL=0
MOVL C00506 V=800.0 PL=0
MOVL C00507 V=800.0 PL=0
MOVL C00508 V=800.0 PL=0
MOVL C00509 V=800.0 PL=0
MOVL C00510 V=800.0 PL=0
MOVL C00511 V=800.0 PL=0
MOVL C00512 V=800.0 PL=0
MOVL C00513 V=800.0 PL=0
MOVL C00514 V=800.0 PL=0
MOVL C00515 V=800.0 PL=0
MOVL C00516 V=800.0 PL=0
MOVL C00517 V=800.0 PL=0
MOVL C00518 V=800.0 PL=0
MOVL C00519 V=800.0 PL=0
MOVL C00520 V=800.0 PL=0
MOVL C00521 V=800.0 PL=0
MOVL C00522 V=800.0 PL=0
MOVL C00523 V=800.0 PL=0
MOVL C00524 V=800.0 PL=0
MOVL C00525 V=800.0 PL=0
MOVL C00526 V=800.0 PL=0
MOVL C00527 V=800.0 PL=0
MOVL C00528 V=800.0 PL=0
MOVL C00529 V=800.0 PL=0
MOVL C00530 V=800.0 PL=0
MOVL C00531 V=800.0 PL=0
MOVL C00532 V=800.0 PL=0
MOVL C00533 V=800.0 PL=0
MOVL C00534 V=800.0 PL=0
MOVL C00535 V=800.0 PL=0
MOVL C00536 V=800.0 PL=0
MOVL C00537 V=800.0 PL=0
MOVL C00538 V=800.0 PL=0
MOVL C00539 V=800.0 PL=0
MOVL C00540 V=800.0 PL=0
MOVL C00541 V=800.0 PL=0
MOVL C00542 V=800.0 PL=0
MOVL C00543 V=800.0 PL=0
MOVL C00544 V=800.0 PL=0
MOVL C00545 V=800.0 PL=0
MOVL C00546 V=800.0 PL=0
MOVL C00547 V=800.0 PL=0
MOVL C00548 V=800.0 PL=0
MOVL C00549 V=800.0 PL=0
MOVL C00550 V=800.0 PL=0
MOVL C00551 V=800.0 PL=0
MOVL C00552 V=800.0 PL=0
MOVL C00553 V=800.0 PL=0
MOVL C00554 V=800.0 PL=0
MOVL C00555 V=800.0 PL=0
MOVL C00556 V=800.0 PL=0
MOVL C00557 V=800.0 PL=0
MOVL C00558 V=800.0 PL=0
MOVL C00559 V=800.0 PL=0
MOVL C00560 V=800.0 PL=0
MOVL C00561 V=800.0 PL=0
MOVL C00562 V=800.0 PL=0
MOVL C00563 V=800.0 PL=0
MOVL C00564 V=800.0 PL=0
MOVL C00565 V=800.0 PL=0
MOVL C00566 V=800.0 PL=0
MOVL C00567 V=800.0 PL=0
MOVL C00568 V=800.0 PL=0
MOVL C00569 V=800.0 PL=0
MOVL C00570 V=800.0 PL=0
MOVL C00571 V=800.0 PL=0
MOVL C00572 V=800.0 PL=0
MOVL C00573 V=800.0 PL=0
MOVL C00574 V=800.0 PL=0
MOVL C00575 V=800.0 PL=0
MOVL C00576 V=800.0 PL=0
MOVL C00577 V=800.0 PL=0
MOVL C00578 V=800.0 PL=0
MOVL C00579 V=800.0 PL=0
MOVL C00580 V=800.0 PL=0
MOVL C00581 V=800.0 PL=0
MOVL C00582 V=800.0 PL=0
MOVL C00583 V=800.0 PL=0
MOVL C00584 V=800.0 PL=0
MOVL C00585 V=800.0 PL=0
MOVL C00586 V=800.0 PL=0
MOVL C00587 V=800.0 PL=0
MOVL C00588 V=800.0 PL=0
MOVL C00589 V=800.0 PL=0
MOVL C00590 V=800.0 PL=0
MOVL C00591 V=800.0 PL=0
MOVL C00592 V=800.0 PL=0
MOVL C00593 V=800.0 PL=0
MOVL C00594 V=800.0 PL=0
MOVL C00595 V=800.0 PL=0
MOVL C00596 V=800.0 PL=0
MOVL C00597 V=800.0 PL=0
MOVL C00598 V=800.0 PL=0
MOVL C00599 V=800.0 PL=0
MOVL C00600 V=800.0 PL=0
MOVL C00601 V=800.0 PL=0
MOVL C00602 V=800.0 PL=0
MOVL C00603 V=800.0 PL=0
MOVL C00604 V=800.0 PL=0
MOVL C00605 V=800.0 PL=0
MOVL C00606 V=800.0 PL=0
MOVL C00607 V=800.0 PL=0
MOVL C00608 V=800.0 PL=0
MOVL C00609 V=800.0 PL=0
MOVL C00610 V=800.0 PL=0
MOVL C00611 V=800.0 PL=0
MOVL C00612 V=800.0 PL=0
MOVL C00613 V=800.0 PL=0
MOVL C00614 V=800.0 PL=0
MOVL C00615 V=800.0 PL=0
MOVL C00616 V=800.0 PL=0
MOVL C00617 V=800.0 PL=0
MOVL C00618 V=800.0 PL=0
MOVL C00619 V=800.0 PL=0
MOVL C00620 V=800.0 PL=0
MOVL C00621 V=800.0 PL=0
MOVL C00622 V=800.0 PL=0
MOVL C00623 V=800.0 PL=0
MOVL C00624 V=800.0 PL=0
MOVL C00625 V=800.0 PL=0
MOVL C00626 V=800.0 PL=0
MOVL C00627 V=800.0 PL=0
MOVL C00628 V=800.0 PL=0
MOVL C00629 V=800.0 PL=0
MOVL C00630 V=800.0 PL=0
MOVL C00631 V=800.0 PL=0
MOVL C00632 V=800.0 PL=0
MOVL C00633 V=800.0 PL=0
MOVL C00634 V=800.0 PL=0
MOVL C00635 V=800.0 PL=0
MOVL C00636 V=800.0 PL=0
MOVL C00637 V=800.0 PL=0
MOVL C00638 V=800.0 PL=0
MOVL C00639 V=800.0 PL=0
MOVL C00640 V=800.0 PL=0
MOVL C00641 V=800.0 PL=0
MOVL C00642 V=800.0 PL=0
MOVL C00643 V=800.0 PL=0
MOVL C00644 V=800.0 PL=0
MOVL C00645 V=800.0 PL=0
MOVL C00646 V=800.0 PL=0
MOVL C00647 V=800.0 PL=0
MOVL C00648 V=800.0 PL=0
MOVL C00649 V=800.0 PL=0
MOVL C00650 V=800.0 PL=0
MOVL C00651 V=800.0 PL=0
MOVL C00652 V=800.0 PL=0
MOVL C00653 V=800.0 PL=0
MOVL C00654 V=800.0 PL=0
MOVL C00655 V=800.0 PL=0
MOVL C00656 V=800.0 PL=0
MOVL C00657 V=800.0 PL=0
MOVL C00658 V=800.0 PL=0
MOVL C00659 V=800.0 PL=0
MOVL C00660 V=800.0 PL=0
MOVL C00661 V=800.0 PL=0
MOVL C00662 V=800.0 PL=0
MOVL C00663 V=800.0 PL=0
MOVL C00664 V=800.0 PL=0
MOVL C00665 V=800.0 PL=0
MOVL C00666 V=800.0 PL=0
MOVL C00667 V=800.0 PL=0
MOVL C00668 V=800.0 PL=0
MOVL C00669 V=800.0 PL=0
MOVL C00670 V=800.0 PL=0
MOVL C00671 V=800.0 PL=0
MOVL C00672 V=800.0 PL=0
MOVL C00673 V=800.0 PL=0
MOVL C00674 V=800.0 PL=0
MOVL C00675 V=800.0 PL=0
MOVL C00676 V=800.0 PL=0
MOVL C00677 V=800.0 PL=0
MOVL C00678 V=800.0 PL=0
MOVL C00679 V=800.0 PL=0
MOVL C00680 V=800.0 PL=0
MOVL C00681 V=800.0 PL=0
MOVL C00682 V=800.0 PL=0
MOVL C00683 V=800.0 PL=0
MOVL C00684 V=800.0 PL=0
MOVL C00685 V=800.0 PL=0
MOVL C00686 V=800.0 PL=0
MOVL C00687 V=800.0 PL=0
MOVL C00688 V=800.0 PL=0
MOVL C00689 V=800.0 PL=0
MOVL C00690 V=800.0 PL=0
MOVL C00691 V=800.0 PL=0
MOVL C00692 V=800.0 PL=0
MOVL C00693 V=800.0 PL=0
MOVL C00694 V=800.0 PL=0
MOVL C00695 V=800.0 PL=0
MOVL C00696 V=800.0 PL=0
MOVL C00697 V=800.0 PL=0
MOVL C00698 V=800.0 PL=0
MOVL C00699 V=800.0 PL=0
MOVL C00700 V=800.0 PL=0
MOVL C00701 V=800.0 PL=0
MOVL C00702 V=800.0 PL=0
MOVL C00703 V=800.0 PL=0
MOVL C00704 V=800.0 PL=0
MOVL C00705 V=800.0 PL=0
MOVL C00706 V=800.0 PL=0
MOVL C00707 V=800.0 PL=0
MOVL C00708 V=800.0 PL=0
MOVL C00709 V=800.0 PL=0
MOVL C00710 V=800.0 PL=0
MOVL C00711 V=800.0 PL=0
MOVL C00712 V=800.0 PL=0
MOVL C00713 V=800.0 PL=0
MOVL C00714 V=800.0 PL=0
MOVL C00715 V=800.0 PL=0
MOVL C00716 V=800.0 PL=0
MOVL C00717 V=800.0 PL=0
MOVL C00718 V=800.0 PL=0
MOVL C00719 V=800.0 PL=0
MOVL C00720 V=800.0 PL=0
MOVL C00721 V=800.0 PL=0
MOVL C00722 V=800.0 PL=0
MOVL C00723 V=800.0 PL=0
MOVL C00724 V=800.0 PL=0
MOVL C00725 V=800.0 PL=0
MOVL C00726 V=800.0 PL=0
MOVL C00727 V=800.0 PL=0
MOVL C00728 V=800.0 PL=0
MOVL C00729 V=800.0 PL=0
MOVL C00730 V=800.0 PL=0
MOVL C00731 V=800.0 PL=0
MOVL C00732 V=800.0 PL=0
MOVL C00733 V=800.0 PL=0
MOVL C00734 V=800.0 PL=0
MOVL C00735 V=800.0 PL=0
MOVL C00736 V=800.0 PL=0
MOVL C00737 V=800.0 PL=0
MOVL C00738 V=800.0 PL=0
MOVL C00739 V=800.0 PL=0
MOVL C00740 V=800.0 PL=0
MOVL C00741 V=800.0 PL=0
MOVL C00742 V=800.0 PL=0
MOVL C00743 V=800.0 PL=0
MOVL C00744 V=800.0 PL=0
MOVL C00745 V=800.0 PL=0
MOVL C00746 V=800.0 PL=0
MOVL C00747 V=800.0 PL=0
MOVL C00748 V=800.0 PL=0
MOVL C00749 V=800.0 PL=0
MOVL C00750 V=800.0 PL=0
MOVL C00751 V=800.0 PL=0
MOVL C00752 V=800.0 PL=0
MOVL C00753 V=800.0 PL=0
MOVL C00754 V=800.0 PL=0
MOVL C00755 V=800.0 PL=0
MOVL C00756 V=800.0 PL=0
MOVL C00757 V=800.0 PL=0
MOVL C00758 V=800.0 PL=0
MOVL C00759 V=800.0 PL=0
MOVL C00760 V=800.0 PL=0
MOVL C00761 V=800.0 PL=0
MOVL C00762 V=800.0 PL=0
MOVL C00763 V=800.0 PL=0
MOVL C00764 V=800.0 PL=0
MOVL C00765 V=800.0 PL=0
MOVL C00766 V=800.0 PL=0
MOVL C00767 V=800.0 PL=0
MOVL C00768 V=800.0 PL=0
MOVL C00769 V=800.0 PL=0
MOVL C00770 V=800.0 PL=0
MOVL C00771 V=800.0 PL=0
MOVL C00772 V=800.0 PL=0
MOVL C00773 V=800.0 PL=0
MOVL C00774 V=800.0 PL=0
MOVL C00775 V=800.0 PL=0
MOVL C00776 V=800.0 PL=0
MOVL C00777 V=800.0 PL=0
MOVL C00778 V=800.0 PL=0
MOVL C00779 V=800.0 PL=0
MOVL C00780 V=800.0 PL=0
MOVL C00781 V=800.0 PL=0
MOVL C00782 V=800.0 PL=0
MOVL C00783 V=800.0 PL=0
MOVL C00784 V=800.0 PL=0
MOVL C00785 V=800.0 PL=0
MOVL C00786 V=800.0 PL=0
MOVL C00787 V=800.0 PL=0
MOVL C00788 V=800.0 PL=0
MOVL C00789 V=800.0 PL=0
MOVL C00790 V=800.0 PL=0
MOVL C00791 V=800.0 PL=0
MOVL C00792 V=800.0 PL=0
MOVL C00793 V=800.0 PL=0
MOVL C00794 V=800.0 PL=0
MOVL C00795 V=800.0 PL=0
MOVL C00796 V=800.0 PL=0
MOVL C00797 V=800.0 PL=0
MOVL C00798 V=800.0 PL=0
MOVL C00799 V=800.0 PL=0
MOVL C00800 V=800.0 PL=0
MOVL C00801 V=800.0 PL=0
MOVL C00802 V=800.0 PL=0
MOVL C00803 V=800.0 PL=0
MOVL C00804 V=800.0 PL=0
MOVL C00805 V=800.0 PL=0
MOVL C00806 V=800.0 PL=0
MOVL C00807 V=800.0 PL=0
MOVL C00808 V=800.0 PL=0
MOVL C00809 V=800.0 PL=0
MOVL C00810 V=800.0 PL=0
MOVL C00811 V=800.0 PL=0
MOVL C00812 V=800.0 PL=0
MOVL C00813 V=800.0 PL=0
MOVL C00814 V=800.0 PL=0
MOVL C00815 V=800.0 PL=0
MOVL C00816 V=800.0 PL=0
MOVL C00817 V=800.0 PL=0
MOVL C00818 V=800.0 PL=0
MOVL C00819 V=800.0 PL=0
MOVL C00820 V=800.0 PL=0
MOVL C00821 V=800.0 PL=0
MOVL C00822 V=800.0 PL=0
MOVL C00823 V=800.0 PL=0
MOVL C00824 V=800.0 PL=0
MOVL C00825 V=800.0 PL=0
MOVL C00826 V=800.0 PL=0
MOVL C00827 V=800.0 PL=0
MOVL C00828 V=800.0 PL=0
MOVL C00829 V=800.0 PL=0
MOVL C00830 V=800.0 PL=0
MOVL C00831 V=800.0 PL=0
MOVL C00832 V=800.0 PL=0
MOVL C00833 V=800.0 PL=0
MOVL C00834 V=800.0 PL=0
MOVL C00835 V=800.0 PL=0
MOVL C00836 V=800.0 PL=0
MOVL C00837 V=800.0 PL=0
MOVL C00838 V=800.0 PL=0
MOVL C00839 V=800.0 PL=0
MOVL C00840 V=800.0 PL=0
MOVL C00841 V=800.0 PL=0
MOVL C00842 V=800.0 PL=0
MOVL C00843 V=800.0 PL=0
MOVL C00844 V=800.0 PL=0
MOVL C00845 V=800.0 PL=0
MOVL C00846 V=800.0 PL=0
MOVL C00847 V=800.0 PL=0
MOVL C00848 V=800.0 PL=0
MOVL C00849 V=800.0 PL=0
MOVL C00850 V=800.0 PL=0
MOVL C00851 V=800.0 PL=0
MOVL C00852 V=800.0 PL=0
MOVL C00853 V=800.0 PL=0
MOVL C00854 V=800.0 PL=0
MOVL C00855 V=800.0 PL=0
MOVL C00856 V=800.0 PL=0
MOVL C00857 V=800.0 PL=0
MOVL C00858 V=800.0 PL=0
MOVL C00859 V=800.0 PL=0
MOVL C00860 V=800.0 PL=0
MOVL C00861 V=800.0 PL=0
MOVL C00862 V=800.0 PL=0
MOVL C00863 V=800.0 PL=0
MOVL C00864 V=800.0 PL=0
MOVL C00865 V=800.0 PL=0
MOVL C00866 V=800.0 PL=0
MOVL C00867 V=800.0 PL=0
MOVL C00868 V=800.0 PL=0
MOVL C00869 V=800.0 PL=0
MOVL C00870 V=800.0 PL=0
MOVL C00871 V=800.0 PL=0
MOVL C00872 V=800.0 PL=0
MOVL C00873 V=800.0 PL=0
MOVL C00874 V=800.0 PL=0
MOVL C00875 V=800.0 PL=0
MOVL C00876 V=800.0 PL=0
MOVL C00877 V=800.0 PL=0
MOVL C00878 V=800.0 PL=0
MOVL C00879 V=800.0 PL=0
MOVL C00880 V=800.0 PL=0
MOVL C00881 V=800.0 PL=0
MOVL C00882 V=800.0 PL=0
MOVL C00883 V=800.0 PL=0
MOVL C00884 V=800.0 PL=0
MOVL C00885 V=800.0 PL=0
MOVL C00886 V=800.0 PL=0
MOVL C00887 V=800.0 PL=0
MOVL C00888 V=800.0 PL=0
MOVL C00889 V=800.0 PL=0
MOVL C00890 V=800.0 PL=0
MOVL C00891 V=800.0 PL=0
MOVL C00892 V=800.0 PL=0
MOVL C00893 V=800.0 PL=0
MOVL C00894 V=800.0 PL=0
MOVL C00895 V=800.0 PL=0
MOVL C00896 V=800.0 PL=0
MOVL C00897 V=800.0 PL=0
MOVL C00898 V=800.0 PL=0
MOVL C00899 V=800.0 PL=0
MOVL C00900 V=800.0 PL=0
MOVL C00901 V=800.0 PL=0
MOVL C00902 V=800.0 PL=0
MOVL C00903 V=800.0 PL=0
MOVL C00904 V=800.0 PL=0
MOVL C00905 V=800.0 PL=0
MOVL C00906 V=800.0 PL=0
MOVL C00907 V=800.0 PL=0
MOVL C00908 V=800.0 PL=0
MOVL C00909 V=800.0 PL=0
MOVL C00910 V=800.0 PL=0
MOVL C00911 V=800.0 PL=0
MOVL C00912 V=800.0 PL=0
MOVL C00913 V=800.0 PL=0
MOVL C00914 V=800.0 PL=0
MOVL C00915 V=800.0 PL=0
MOVL C00916 V=800.0 PL=0
MOVL C00917 V=800.0 PL=0
MOVL C00918 V=800.0 PL=0
MOVL C00919 V=800.0 PL=0
MOVL C00920 V=800.0 PL=0
MOVL C00921 V=800.0 PL=0
MOVL C00922 V=800.0 PL=0
MOVL C00923 V=800.0 PL=0
MOVL C00924 V=800.0 PL=0
MOVL C00925 V=800.0 PL=0
MOVL C00926 V=800.0 PL=0
MOVL C00927 V=800.0 PL=0
MOVL C00928 V=800.0 PL=0
MOVL C00929 V=800.0 PL=0
MOVL C00930 V=800.0 PL=0
MOVL C00931 V=800.0 PL=0
MOVL C00932 V=800.0 PL=0
MOVL C00933 V=800.0 PL=0
MOVL C00934 V=800.0 PL=0
MOVL C00935 V=800.0 PL=0
MOVL C00936 V=800.0 PL=0
MOVL C00937 V=800.0 PL=0
MOVL C00938 V=800.0 PL=0
MOVL C00939 V=800.0 PL=0
MOVL C00940 V=800.0 PL=0
MOVL C00941 V=800.0 PL=0
MOVL C00942 V=800.0 PL=0
MOVL C00943 V=800.0 PL=0
MOVL C00944 V=800.0 PL=0
MOVL C00945 V=800.0 PL=0
MOVL C00946 V=800.0 PL=0
MOVL C00947 V=800.0 PL=0
MOVL C00948 V=800.0 PL=0
MOVL C00949 V=800.0 PL=0
MOVL C00950 V=800.0 PL=0
MOVL C00951 V=800.0 PL=0
MOVL C00952 V=800.0 PL=0
MOVL C00953 V=800.0 PL=0
MOVL C00954 V=800.0 PL=0
MOVL C00955 V=800.0 PL=0
MOVL C00956 V=800.0 PL=0
MOVL C00957 V=800.0 PL=0
MOVL C00958 V=800.0 PL=0
MOVL C00959 V=800.0 PL=0
MOVL C00960 V=800.0 PL=0
MOVL C00961 V=800.0 PL=0
MOVL C00962 V=800.0 PL=0
MOVL C00963 V=800.0 PL=0
MOVL C00964 V=800.0 PL=0
MOVL C00965 V=800.0 PL=0
MOVL C00966 V=800.0 PL=0
MOVL C00967 V=800.0 PL=0
MOVL C00968 V=800.0 PL=0
MOVL C00969 V=800.0 PL=0
MOVL C00970 V=800.0 PL=0
MOVL C00971 V=800.0 PL=0
MOVL C00972 V=800.0 PL=0
MOVL C00973 V=800.0 PL=0
MOVL C00974 V=800.0 PL=0
MOVL C00975 V=800.0 PL=0
MOVL C00976 V=800.0 PL=0
MOVL C00977 V=800.0 PL=0
MOVL C00978 V=800.0 PL=0
MOVL C00979 V=800.0 PL=0
MOVL C00980 V=800.0 PL=0
MOVL C00981 V=800.0 PL=0
MOVL C00982 V=800.0 PL=0
MOVL C00983 V=800.0 PL=0
MOVL C00984 V=800.0 PL=0
MOVL C00985 V=800.0 PL=0
MOVL C00986 V=800.0 PL=0
MOVL C00987 V=800.0 PL=0
MOVL C00988 V=800.0 PL=0
MOVL C00989 V=800.0 PL=0
MOVL C00990 V=800.0 PL=0
MOVL C00991 V=800.0 PL=0
MOVL C00992 V=800.0 PL=0
MOVL C00993 V=800.0 PL=0
MOVL C00994 V=800.0 PL=0
MOVL C00995 V=800.0 PL=0
MOVL C00996 V=800.0 PL=0
MOVL C00997 V=800.0 PL=0
MOVL C00998 V=800.0 PL=0
MOVL C00999 V=800.0 PL=0
MOVL C01000 V=800.0 PL=0
MOVL C01001 V=800.0 PL=0
MOVL C01002 V=800.0 PL=0
MOVL C01003 V=800.0 PL=0
MOVL C01004 V=800.0 PL=0
MOVL C01005 V=800.0 PL=0
MOVL C01006 V=800.0 PL=0
MOVL C01007 V=800.0 PL=0
MOVL C01008 V=800.0 PL=0
MOVL C01009 V=800.0 PL=0
MOVL C01010 V=800.0 PL=0
MOVL C01011 V=800.0 PL=0
MOVL C01012 V=800.0 PL=0
MOVL C01013 V=800.0 PL=0
MOVL C01014 V=800.0 PL=0
MOVL C01015 V=800.0 PL=0
MOVL C01016 V=800.0 PL=0
MOVL C01017 V=800.0 PL=0
MOVL C01018 V=800.0 PL=0
MOVL C01019 V=800.0 PL=0
MOVL C01020 V=800.0 PL=0
MOVL C01021 V=800.0 PL=0
MOVL C01022 V=800.0 PL=0
MOVL C01023 V=800.0 PL=0
MOVL C01024 V=800.0 PL=0
MOVL C01025 V=800.0 PL=0
MOVL C01026 V=800.0 PL=0
MOVL C01027 V=800.0 PL=0
MOVL C01028 V=800.0 PL=0
MOVL C01029 V=800.0 PL=0
MOVL C01030 V=800.0 PL=0
MOVL C01031 V=800.0 PL=0
MOVL C01032 V=800.0 PL=0
MOVL C01033 V=800.0 PL=0
MOVL C01034 V=800.0 PL=0
MOVL C01035 V=800.0 PL=0
MOVL C01036 V=800.0 PL=0
MOVL C01037 V=800.0 PL=0
MOVL C01038 V=800.0 PL=0
MOVL C01039 V=800.0 PL=0
MOVL C01040 V=800.0 PL=0
MOVL C01041 V=800.0 PL=0
MOVL C01042 V=800.0 PL=0
MOVL C01043 V=800.0 PL=0
MOVL C01044 V=800.0 PL=0
MOVL C01045 V=800.0 PL=0
MOVL C01046 V=800.0 PL=0
MOVL C01047 V=800.0 PL=0
MOVL C01048 V=800.0 PL=0
MOVL C01049 V=800.0 PL=0
MOVL C01050 V=800.0 PL=0
MOVL C01051 V=800.0 PL=0
MOVL C01052 V=800.0 PL=0
MOVL C01053 V=800.0 PL=0
MOVL C01054 V=800.0 PL=0
MOVL C01055 V=800.0 PL=0
MOVL C01056 V=800.0 PL=0
MOVL C01057 V=800.0 PL=0
MOVL C01058 V=800.0 PL=0
MOVL C01059 V=800.0 PL=0
MOVL C01060 V=800.0 PL=0
MOVL C01061 V=800.0 PL=0
MOVL C01062 V=800.0 PL=0
MOVL C01063 V=800.0 PL=0
MOVL C01064 V=800.0 PL=0
MOVL C01065 V=800.0 PL=0
MOVL C01066 V=800.0 PL=0
MOVL C01067 V=800.0 PL=0
MOVL C01068 V=800.0 PL=0
MOVL C01069 V=800.0 PL=0
MOVL C01070 V=800.0 PL=0
MOVL C01071 V=800.0 PL=0
MOVL C01072 V=800.0 PL=0
MOVL C01073 V=800.0 PL=0
MOVL C01074 V=800.0 PL=0
MOVL C01075 V=800.0 PL=0
MOVL C01076 V=800.0 PL=0
MOVL C01077 V=800.0 PL=0
MOVL C01078 V=800.0 PL=0
MOVL C01079 V=800.0 PL=0
MOVL C01080 V=800.0 PL=0
MOVL C01081 V=800.0 PL=0
MOVL C01082 V=800.0 PL=0
MOVL C01083 V=800.0 PL=0
MOVL C01084 V=800.0 PL=0
MOVL C01085 V=800.0 PL=0
MOVL C01086 V=800.0 PL=0
MOVL C01087 V=800.0 PL=0
MOVL C01088 V=800.0 PL=0
MOVL C01089 V=800.0 PL=0
MOVL C01090 V=800.0 PL=0
MOVL C01091 V=800.0 PL=0
MOVL C01092 V=800.0 PL=0
MOVL C01093 V=800.0 PL=0
MOVL C01094 V=800.0 PL=0
MOVL C01095 V=800.0 PL=0
MOVL C01096 V=800.0 PL=0
MOVL C01097 V=800.0 PL=0
MOVL C01098 V=800.0 PL=0
MOVL C01099 V=800.0 PL=0
MOVL C01100 V=800.0 PL=0
MOVL C01101 V=800.0 PL=0
MOVL C01102 V=800.0 PL=0
MOVL C01103 V=800.0 PL=0
MOVL C01104 V=800.0 PL=0
MOVL C01105 V=800.0 PL=0
MOVL C01106 V=800.0 PL=0
MOVL C01107 V=800.0 PL=0
MOVL C01108 V=800.0 PL=0
MOVL C01109 V=800.0 PL=0
MOVL C01110 V=800.0 PL=0
MOVL C01111 V=800.0 PL=0
MOVL C01112 V=800.0 PL=0
MOVL C01113 V=800.0 PL=0
MOVL C01114 V=800.0 PL=0
MOVL C01115 V=800.0 PL=0
MOVL C01116 V=800.0 PL=0
MOVL C01117 V=800.0 PL=0
MOVL C01118 V=800.0 PL=0
MOVL C01119 V=800.0 PL=0
MOVL C01120 V=800.0 PL=0
MOVL C01121 V=800.0 PL=0
MOVL C01122 V=800.0 PL=0
MOVL C01123 V=800.0 PL=0
MOVL C01124 V=800.0 PL=0
MOVL C01125 V=800.0 PL=0
MOVL C01126 V=800.0 PL=0
MOVL C01127 V=800.0 PL=0
MOVL C01128 V=800.0 PL=0
MOVL C01129 V=800.0 PL=0
MOVL C01130 V=800.0 PL=0
MOVL C01131 V=800.0 PL=0
MOVL C01132 V=800.0 PL=0
MOVL C01133 V=800.0 PL=0
MOVL C01134 V=800.0 PL=0
MOVL C01135 V=800.0 PL=0
MOVL C01136 V=800.0 PL=0
MOVL C01137 V=800.0 PL=0
MOVL C01138 V=800.0 PL=0
MOVL C01139 V=800.0 PL=0
MOVL C01140 V=800.0 PL=0
MOVL C01141 V=800.0 PL=0
MOVL C01142 V=800.0 PL=0
MOVL C01143 V=800.0 PL=0
MOVL C01144 V=800.0 PL=0
MOVL C01145 V=800.0 PL=0
MOVL C01146 V=800.0 PL=0
MOVL C01147 V=800.0 PL=0
MOVL C01148 V=800.0 PL=0
MOVL C01149 V=800.0 PL=0
MOVL C01150 V=800.0 PL=0
MOVL C01151 V=800.0 PL=0
MOVL C01152 V=800.0 PL=0
MOVL C01153 V=800.0 PL=0
MOVL C01154 V=800.0 PL=0
MOVL C01155 V=800.0 PL=0
MOVL C01156 V=800.0 PL=0
MOVL C01157 V=800.0 PL=0
MOVL C01158 V=800.0 PL=0
MOVL C01159 V=800.0 PL=0
MOVL C01160 V=800.0 PL=0
MOVL C01161 V=800.0 PL=0
MOVL C01162 V=800.0 PL=0
MOVL C01163 V=800.0 PL=0
MOVL C01164 V=800.0 PL=0
MOVL C01165 V=800.0 PL=0
MOVL C01166 V=800.0 PL=0
MOVL C01167 V=800.0 PL=0
MOVL C01168 V=800.0 PL=0
MOVL C01169 V=800.0 PL=0
MOVL C01170 V=800.0 PL=0
MOVL C01171 V=800.0 PL=0
MOVL C01172 V=800.0 PL=0
MOVL C01173 V=800.0 PL=0
MOVL C01174 V=800.0 PL=0
MOVL C01175 V=800.0 PL=0
MOVL C01176 V=800.0 PL=0
MOVL C01177 V=800.0 PL=0
MOVL C01178 V=800.0 PL=0
MOVL C01179 V=800.0 PL=0
MOVL C01180 V=800.0 PL=0
MOVL C01181 V=800.0 PL=0
MOVL C01182 V=800.0 PL=0
MOVL C01183 V=800.0 PL=0
MOVL C01184 V=800.0 PL=0
MOVL C01185 V=800.0 PL=0
MOVL C01186 V=800.0 PL=0
MOVL C01187 V=800.0 PL=0
MOVL C01188 V=800.0 PL=0
MOVL C01189 V=800.0 PL=0
MOVL C01190 V=800.0 PL=0
MOVL C01191 V=800.0 PL=0
MOVL C01192 V=800.0 PL=0
MOVL C01193 V=800.0 PL=0
MOVL C01194 V=800.0 PL=0
MOVL C01195 V=800.0 PL=0
MOVL C01196 V=800.0 PL=0
MOVL C01197 V=800.0 PL=0
MOVL C01198 V=800.0 PL=0
MOVL C01199 V=800.0 PL=0
MOVL C01200 V=800.0 PL=0
MOVL C01201 V=800.0 PL=0
MOVL C01202 V=800.0 PL=0
MOVL C01203 V=800.0 PL=0
MOVL C01204 V=800.0 PL=0
MOVL C01205 V=800.0 PL=0
MOVL C01206 V=800.0 PL=0
MOVL C01207 V=800.0 PL=0
MOVL C01208 V=800.0 PL=0
MOVL C01209 V=800.0 PL=0
MOVL C01210 V=800.0 PL=0
MOVL C01211 V=800.0 PL=0
MOVL C01212 V=800.0 PL=0
MOVL C01213 V=800.0 PL=0
MOVL C01214 V=800.0 PL=0
MOVL C01215 V=800.0 PL=0
MOVL C01216 V=800.0 PL=0
MOVL C01217 V=800.0 PL=0
MOVL C01218 V=800.0 PL=0
MOVL C01219 V=800.0 PL=0
MOVL C01220 V=800.0 PL=0
MOVL C01221 V=800.0 PL=0
MOVL C01222 V=800.0 PL=0
MOVL C01223 V=800.0 PL=0
MOVL C01224 V=800.0 PL=0
MOVL C01225 V=800.0 PL=0
MOVL C01226 V=800.0 PL=0
MOVL C01227 V=800.0 PL=0
MOVL C01228 V=800.0 PL=0
MOVL C01229 V=800.0 PL=0
MOVL C01230 V=800.0 PL=0
MOVL C01231 V=800.0 PL=0
MOVL C01232 V=800.0 PL=0
MOVL C01233 V=800.0 PL=0
MOVL C01234 V=800.0 PL=0
MOVL C01235 V=800.0 PL=0
MOVL C01236 V=800.0 PL=0
MOVL C01237 V=800.0 PL=0
MOVL C01238 V=800.0 PL=0
MOVL C01239 V=800.0 PL=0
MOVL C01240 V=800.0 PL=0
MOVL C01241 V=800.0 PL=0
MOVL C01242 V=800.0 PL=0
MOVL C01243 V=800.0 PL=0
MOVL C01244 V=800.0 PL=0
MOVL C01245 V=800.0 PL=0
MOVL C01246 V=800.0 PL=0
MOVL C01247 V=800.0 PL=0
MOVL C01248 V=800.0 PL=0
MOVL C01249 V=800.0 PL=0
MOVL C01250 V=800.0 PL=0
MOVL C01251 V=800.0 PL=0
MOVL C01252 V=800.0 PL=0
MOVL C01253 V=800.0 PL=0
MOVL C01254 V=800.0 PL=0
MOVL C01255 V=800.0 PL=0
MOVL C01256 V=800.0 PL=0
MOVL C01257 V=800.0 PL=0
MOVL C01258 V=800.0 PL=0
MOVL C01259 V=800.0 PL=0
MOVL C01260 V=800.0 PL=0
MOVL C01261 V=800.0 PL=0
MOVL C01262 V=800.0 PL=0
MOVL C01263 V=800.0 PL=0
MOVL C01264 V=800.0 PL=0
MOVL C01265 V=800.0 PL=0
MOVL C01266 V=800.0 PL=0
MOVL C01267 V=800.0 PL=0
MOVL C01268 V=800.0 PL=0
MOVL C01269 V=800.0 PL=0
MOVL C01270 V=800.0 PL=0
MOVL C01271 V=800.0 PL=0
MOVL C01272 V=800.0 PL=0
MOVL C01273 V=800.0 PL=0
MOVL C01274 V=800.0 PL=0
MOVL C01275 V=800.0 PL=0
MOVL C01276 V=800.0 PL=0
MOVL C01277 V=800.0 PL=0
MOVL C01278 V=800.0 PL=0
MOVL C01279 V=800.0 PL=0
MOVL C01280 V=800.0 PL=0
MOVL C01281 V=800.0 PL=0
MOVL C01282 V=800.0 PL=0
MOVL C01283 V=800.0 PL=0
MOVL C01284 V=800.0 PL=0
MOVL C01285 V=800.0 PL=0
MOVL C01286 V=800.0 PL=0
MOVL C01287 V=800.0 PL=0
MOVL C01288 V=800.0 PL=0
MOVL C01289 V=800.0 PL=0
MOVL C01290 V=800.0 PL=0
MOVL C01291 V=800.0 PL=0
MOVL C01292 V=800.0 PL=0
MOVL C01293 V=800.0 PL=0
MOVL C01294 V=800.0 PL=0
MOVL C01295 V=800.0 PL=0
MOVL C01296 V=800.0 PL=0
MOVL C01297 V=800.0 PL=0
MOVL C01298 V=800.0 PL=0
MOVL C01299 V=800.0 PL=0
MOVL C01300 V=800.0 PL=0
MOVL C01301 V=800.0 PL=0
MOVL C01302 V=800.0 PL=0
MOVL C01303 V=800.0 PL=0
MOVL C01304 V=800.0 PL=0
MOVL C01305 V=800.0 PL=0
MOVL C01306 V=800.0 PL=0
MOVL C01307 V=800.0 PL=0
MOVL C01308 V=800.0 PL=0
MOVL C01309 V=800.0 PL=0
MOVL C01310 V=800.0 PL=0
MOVL C01311 V=800.0 PL=0
MOVL C01312 V=800.0 PL=0
MOVL C01313 V=800.0 PL=0
MOVL C01314 V=800.0 PL=0
MOVL C01315 V=800.0 PL=0
MOVL C01316 V=800.0 PL=0
MOVL C01317 V=800.0 PL=0
MOVL C01318 V=800.0 PL=0
MOVL C01319 V=800.0 PL=0
MOVL C01320 V=800.0 PL=0
MOVL C01321 V=800.0 PL=0
MOVL C01322 V=800.0 PL=0
MOVL C01323 V=800.0 PL=0
MOVL C01324 V=800.0 PL=0
MOVL C01325 V=800.0 PL=0
MOVL C01326 V=800.0 PL=0
MOVL C01327 V=800.0 PL=0
MOVL C01328 V=800.0 PL=0
MOVL C01329 V=800.0 PL=0
MOVL C01330 V=800.0 PL=0
MOVL C01331 V=800.0 PL=0
MOVL C01332 V=800.0 PL=0
MOVL C01333 V=800.0 PL=0
MOVL C01334 V=800.0 PL=0
MOVL C01335 V=800.0 PL=0
MOVL C01336 V=800.0 PL=0
MOVL C01337 V=800.0 PL=0
MOVL C01338 V=800.0 PL=0
MOVL C01339 V=800.0 PL=0
MOVL C01340 V=800.0 PL=0
MOVL C01341 V=800.0 PL=0
MOVL C01342 V=800.0 PL=0
MOVL C01343 V=800.0 PL=0
MOVL C01344 V=800.0 PL=0
MOVL C01345 V=800.0 PL=0
MOVL C01346 V=800.0 PL=0
MOVL C01347 V=800.0 PL=0
MOVL C01348 V=800.0 PL=0
MOVL C01349 V=800.0 PL=0
MOVL C01350 V=800.0 PL=0
MOVL C01351 V=800.0 PL=0
MOVL C01352 V=800.0 PL=0
MOVL C01353 V=800.0 PL=0
MOVL C01354 V=800.0 PL=0
MOVL C01355 V=800.0 PL=0
MOVL C01356 V=800.0 PL=0
MOVL C01357 V=800.0 PL=0
MOVL C01358 V=800.0 PL=0
MOVL C01359 V=800.0 PL=0
MOVL C01360 V=800.0 PL=0
MOVL C01361 V=800.0 PL=0
MOVL C01362 V=800.0 PL=0
MOVL C01363 V=800.0 PL=0
MOVL C01364 V=800.0 PL=0
MOVL C01365 V=800.0 PL=0
MOVL C01366 V=800.0 PL=0
MOVL C01367 V=800.0 PL=0
MOVL C01368 V=800.0 PL=0
MOVL C01369 V=800.0 PL=0
MOVL C01370 V=800.0 PL=0
MOVL C01371 V=800.0 PL=0
MOVL C01372 V=800.0 PL=0
MOVL C01373 V=800.0 PL=0
MOVL C01374 V=800.0 PL=0
MOVL C01375 V=800.0 PL=0
MOVL C01376 V=800.0 PL=0
MOVL C01377 V=800.0 PL=0
MOVL C01378 V=800.0 PL=0
MOVL C01379 V=800.0 PL=0
MOVL C01380 V=800.0 PL=0
MOVL C01381 V=800.0 PL=0
MOVL C01382 V=800.0 PL=0
MOVL C01383 V=800.0 PL=0
MOVL C01384 V=800.0 PL=0
MOVL C01385 V=800.0 PL=0
MOVL C01386 V=800.0 PL=0
MOVL C01387 V=800.0 PL=0
MOVL C01388 V=800.0 PL=0
MOVL C01389 V=800.0 PL=0
MOVL C01390 V=800.0 PL=0
MOVL C01391 V=800.0 PL=0
MOVL C01392 V=800.0 PL=0
MOVL C01393 V=800.0 PL=0
MOVL C01394 V=800.0 PL=0
MOVL C01395 V=800.0 PL=0
MOVL C01396 V=800.0 PL=0
MOVL C01397 V=800.0 PL=0
MOVL C01398 V=800.0 PL=0
MOVL C01399 V=800.0 PL=0
MOVL C01400 V=800.0 PL=0
MOVL C01401 V=800.0 PL=0
MOVL C01402 V=800.0 PL=0
MOVL C01403 V=800.0 PL=0
MOVL C01404 V=800.0 PL=0
MOVL C01405 V=800.0 PL=0
MOVL C01406 V=800.0 PL=0
MOVL C01407 V=800.0 PL=0
MOVL C01408 V=800.0 PL=0
MOVL C01409 V=800.0 PL=0
MOVL C01410 V=800.0 PL=0
MOVL C01411 V=800.0 PL=0
MOVL C01412 V=800.0 PL=0
MOVL C01413 V=800.0 PL=0
MOVL C01414 V=800.0 PL=0
MOVL C01415 V=800.0 PL=0
MOVL C01416 V=800.0 PL=0
MOVL C01417 V=800.0 PL=0
MOVL C01418 V=800.0 PL=0
MOVL C01419 V=800.0 PL=0
MOVL C01420 V=800.0 PL=0
MOVL C01421 V=800.0 PL=0
MOVL C01422 V=800.0 PL=0
MOVL C01423 V=800.0 PL=0
MOVL C01424 V=800.0 PL=0
MOVL C01425 V=800.0 PL=0
MOVL C01426 V=800.0 PL=0
MOVL C01427 V=800.0 PL=0
MOVL C01428 V=800.0 PL=0
MOVL C01429 V=800.0 PL=0
MOVL C01430 V=800.0 PL=0
MOVL C01431 V=800.0 PL=0
MOVL C01432 V=800.0 PL=0
MOVL C01433 V=800.0 PL=0
MOVL C01434 V=800.0 PL=0
MOVL C01435 V=800.0 PL=0
MOVL C01436 V=800.0 PL=0
MOVL C01437 V=800.0 PL=0
MOVL C01438 V=800.0 PL=0
MOVL C01439 V=800.0 PL=0
MOVL C01440 V=800.0 PL=0
MOVL C01441 V=800.0 PL=0
MOVL C01442 V=800.0 PL=0
MOVL C01443 V=800.0 PL=0
MOVL C01444 V=800.0 PL=0
MOVL C01445 V=800.0 PL=0
MOVL C01446 V=800.0 PL=0
MOVL C01447 V=800.0 PL=0
MOVL C01448 V=800.0 PL=0
MOVL C01449 V=800.0 PL=0
MOVL C01450 V=800.0 PL=0
MOVL C01451 V=800.0 PL=0
MOVL C01452 V=800.0 PL=0
MOVL C01453 V=800.0 PL=0
MOVL C01454 V=800.0 PL=0
MOVL C01455 V=800.0 PL=0
MOVL C01456 V=800.0 PL=0
MOVL C01457 V=800.0 PL=0
MOVL C01458 V=800.0 PL=0
MOVL C01459 V=800.0 PL=0
MOVL C01460 V=800.0 PL=0
MOVL C01461 V=800.0 PL=0
MOVL C01462 V=800.0 PL=0
MOVL C01463 V=800.0 PL=0
MOVL C01464 V=800.0 PL=0
MOVL C01465 V=800.0 PL=0
MOVL C01466 V=800.0 PL=0
MOVL C01467 V=800.0 PL=0
MOVL C01468 V=800.0 PL=0
MOVL C01469 V=800.0 PL=0
MOVL C01470 V=800.0 PL=0
MOVL C01471 V=800.0 PL=0
MOVL C01472 V=800.0 PL=0
MOVL C01473 V=800.0 PL=0
MOVL C01474 V=800.0 PL=0
MOVL C01475 V=800.0 PL=0
MOVL C01476 V=800.0 PL=0
MOVL C01477 V=800.0 PL=0
MOVL C01478 V=800.0 PL=0
MOVL C01479 V=800.0 PL=0
MOVL C01480 V=800.0 PL=0
MOVL C01481 V=800.0 PL=0
MOVL C01482 V=800.0 PL=0
MOVL C01483 V=800.0 PL=0
MOVL C01484 V=800.0 PL=0
MOVL C01485 V=800.0 PL=0
MOVL C01486 V=800.0 PL=0
MOVL C01487 V=800.0 PL=0
MOVL C01488 V=800.0 PL=0
MOVL C01489 V=800.0 PL=0
MOVL C01490 V=800.0 PL=0
MOVL C01491 V=800.0 PL=0
MOVL C01492 V=800.0 PL=0
MOVL C01493 V=800.0 PL=0
MOVL C01494 V=800.0 PL=0
MOVL C01495 V=800.0 PL=0
MOVL C01496 V=800.0 PL=0
MOVL C01497 V=800.0 PL=0
MOVL C01498 V=800.0 PL=0
MOVL C01499 V=800.0 PL=0
MOVL C01500 V=800.0 PL=0
MOVL C01501 V=800.0 PL=0
MOVL C01502 V=800.0 PL=0
MOVL C01503 V=800.0 PL=0
MOVL C01504 V=800.0 PL=0
MOVL C01505 V=800.0 PL=0
MOVL C01506 V=800.0 PL=0
MOVL C01507 V=800.0 PL=0
MOVL C01508 V=800.0 PL=0
MOVL C01509 V=800.0 PL=0
MOVL C01510 V=800.0 PL=0
MOVL C01511 V=800.0 PL=0
MOVL C01512 V=800.0 PL=0
MOVL C01513 V=800.0 PL=0
MOVL C01514 V=800.0 PL=0
MOVL C01515 V=800.0 PL=0
MOVL C01516 V=800.0 PL=0
MOVL C01517 V=800.0 PL=0
MOVL C01518 V=800.0 PL=0
MOVL C01519 V=800.0 PL=0
MOVL C01520 V=800.0 PL=0
MOVL C01521 V=800.0 PL=0
MOVL C01522 V=800.0 PL=0
MOVL C01523 V=800.0 PL=0
MOVL C01524 V=800.0 PL=0
MOVL C01525 V=800.0 PL=0
MOVL C01526 V=800.0 PL=0
MOVL C01527 V=800.0 PL=0
MOVL C01528 V=800.0 PL=0
MOVL C01529 V=800.0 PL=0
MOVL C01530 V=800.0 PL=0
MOVL C01531 V=800.0 PL=0
MOVL C01532 V=800.0 PL=0
MOVL C01533 V=800.0 PL=0
MOVL C01534 V=800.0 PL=0
MOVL C01535 V=800.0 PL=0
MOVL C01536 V=800.0 PL=0
MOVL C01537 V=800.0 PL=0
MOVL C01538 V=800.0 PL=0
MOVL C01539 V=800.0 PL=0
MOVL C01540 V=800.0 PL=0
MOVL C01541 V=800.0 PL=0
MOVL C01542 V=800.0 PL=0
MOVL C01543 V=800.0 PL=0
MOVL C01544 V=800.0 PL=0
MOVL C01545 V=800.0 PL=0
MOVL C01546 V=800.0 PL=0
MOVL C01547 V=800.0 PL=0
MOVL C01548 V=800.0 PL=0
MOVL C01549 V=800.0 PL=0
MOVL C01550 V=800.0 PL=0
MOVL C01551 V=800.0 PL=0
MOVL C01552 V=800.0 PL=0
MOVL C01553 V=800.0 PL=0
MOVL C01554 V=800.0 PL=0
MOVL C01555 V=800.0 PL=0
MOVL C01556 V=800.0 PL=0
MOVL C01557 V=800.0 PL=0
MOVL C01558 V=800.0 PL=0
MOVL C01559 V=800.0 PL=0
MOVL C01560 V=800.0 PL=0
MOVL C01561 V=800.0 PL=0
MOVL C01562 V=800.0 PL=0
MOVL C01563 V=800.0 PL=0
MOVL C01564 V=800.0 PL=0
MOVL C01565 V=800.0 PL=0
MOVL C01566 V=800.0 PL=0
MOVL C01567 V=800.0 PL=0
MOVL C01568 V=800.0 PL=0
MOVL C01569 V=800.0 PL=0
MOVL C01570 V=800.0 PL=0
MOVL C01571 V=800.0 PL=0
MOVL C01572 V=800.0 PL=0
MOVL C01573 V=800.0 PL=0
MOVL C01574 V=800.0 PL=0
MOVL C01575 V=800.0 PL=0
MOVL C01576 V=800.0 PL=0
MOVL C01577 V=800.0 PL=0
MOVL C01578 V=800.0 PL=0
MOVL C01579 V=800.0 PL=0
MOVL C01580 V=800.0 PL=0
MOVL C01581 V=800.0 PL=0
MOVL C01582 V=800.0 PL=0
MOVL C01583 V=800.0 PL=0
MOVL C01584 V=800.0 PL=0
MOVL C01585 V=800.0 PL=0
MOVL C01586 V=800.0 PL=0
MOVL C01587 V=800.0 PL=0
MOVL C01588 V=800.0 PL=0
MOVL C01589 V=800.0 PL=0
MOVL C01590 V=800.0 PL=0
MOVL C01591 V=800.0 PL=0
MOVL C01592 V=800.0 PL=0
MOVL C01593 V=800.0 PL=0
MOVL C01594 V=800.0 PL=0
MOVL C01595 V=800.0 PL=0
MOVL C01596 V=800.0 PL=0
MOVL C01597 V=800.0 PL=0
MOVL C01598 V=800.0 PL=0
MOVL C01599 V=800.0 PL=0
MOVL C01600 V=800.0 PL=0
MOVL C01601 V=800.0 PL=0
MOVL C01602 V=800.0 PL=0
MOVL C01603 V=800.0 PL=0
MOVL C01604 V=800.0 PL=0
MOVL C01605 V=800.0 PL=0
MOVL C01606 V=800.0 PL=0
MOVL C01607 V=800.0 PL=0
MOVL C01608 V=800.0 PL=0
MOVL C01609 V=800.0 PL=0
MOVL C01610 V=800.0 PL=0
MOVL C01611 V=800.0 PL=0
MOVL C01612 V=800.0 PL=0
MOVL C01613 V=800.0 PL=0
MOVL C01614 V=800.0 PL=0
MOVL C01615 V=800.0 PL=0
MOVL C01616 V=800.0 PL=0
MOVL C01617 V=800.0 PL=0
MOVL C01618 V=800.0 PL=0
MOVL C01619 V=800.0 PL=0
MOVL C01620 V=800.0 PL=0
MOVL C01621 V=800.0 PL=0
MOVL C01622 V=800.0 PL=0
MOVL C01623 V=800.0 PL=0
MOVL C01624 V=800.0 PL=0
MOVL C01625 V=800.0 PL=0
MOVL C01626 V=800.0 PL=0
MOVL C01627 V=800.0 PL=0
MOVL C01628 V=800.0 PL=0
MOVL C01629 V=800.0 PL=0
MOVL C01630 V=800.0 PL=0
MOVL C01631 V=800.0 PL=0
MOVL C01632 V=800.0 PL=0
MOVL C01633 V=800.0 PL=0
MOVL C01634 V=800.0 PL=0
MOVL C01635 V=800.0 PL=0
MOVL C01636 V=800.0 PL=0
MOVL C01637 V=800.0 PL=0
MOVL C01638 V=800.0 PL=0
MOVL C01639 V=800.0 PL=0
MOVL C01640 V=800.0 PL=0
MOVL C01641 V=800.0 PL=0
MOVL C01642 V=800.0 PL=0
MOVL C01643 V=800.0 PL=0
MOVL C01644 V=800.0 PL=0
MOVL C01645 V=800.0 PL=0
MOVL C01646 V=800.0 PL=0
MOVL C01647 V=800.0 PL=0
MOVL C01648 V=800.0 PL=0
MOVL C01649 V=800.0 PL=0
MOVL C01650 V=800.0 PL=0
MOVL C01651 V=800.0 PL=0
MOVL C01652 V=800.0 PL=0
MOVL C01653 V=800.0 PL=0
MOVL C01654 V=800.0 PL=0
MOVL C01655 V=800.0 PL=0
MOVL C01656 V=800.0 PL=0
MOVL C01657 V=800.0 PL=0
MOVL C01658 V=800.0 PL=0
MOVL C01659 V=800.0 PL=0
MOVL C01660 V=800.0 PL=0
MOVL C01661 V=800.0 PL=0
MOVL C01662 V=800.0 PL=0
MOVL C01663 V=800.0 PL=0
MOVL C01664 V=800.0 PL=0
MOVL C01665 V=800.0 PL=0
MOVL C01666 V=800.0 PL=0
MOVL C01667 V=800.0 PL=0
MOVL C01668 V=800.0 PL=0
MOVL C01669 V=800.0 PL=0
MOVL C01670 V=800.0 PL=0
MOVL C01671 V=800.0 PL=0
MOVL C01672 V=800.0 PL=0
MOVL C01673 V=800.0 PL=0
MOVL C01674 V=800.0 PL=0
MOVL C01675 V=800.0 PL=0
MOVL C01676 V=800.0 PL=0
MOVL C01677 V=800.0 PL=0
MOVL C01678 V=800.0 PL=0
MOVL C01679 V=800.0 PL=0
MOVL C01680 V=800.0 PL=0
MOVL C01681 V=800.0 PL=0
MOVL C01682 V=800.0 PL=0
MOVL C01683 V=800.0 PL=0
MOVL C01684 V=800.0 PL=0
MOVL C01685 V=800.0 PL=0
MOVL C01686 V=800.0 PL=0
MOVL C01687 V=800.0 PL=0
MOVL C01688 V=800.0 PL=0
MOVL C01689 V=800.0 PL=0
MOVL C01690 V=800.0 PL=0
MOVL C01691 V=800.0 PL=0
MOVL C01692 V=800.0 PL=0
MOVL C01693 V=800.0 PL=0
MOVL C01694 V=800.0 PL=0
MOVL C01695 V=800.0 PL=0
MOVL C01696 V=800.0 PL=0
MOVL C01697 V=800.0 PL=0
MOVL C01698 V=800.0 PL=0
MOVL C01699 V=800.0 PL=0
MOVL C01700 V=800.0 PL=0
MOVL C01701 V=800.0 PL=0
MOVL C01702 V=800.0 PL=0
MOVL C01703 V=800.0 PL=0
MOVL C01704 V=800.0 PL=0
MOVL C01705 V=800.0 PL=0
MOVL C01706 V=800.0 PL=0
MOVL C01707 V=800.0 PL=0
MOVL C01708 V=800.0 PL=0
MOVL C01709 V=800.0 PL=0
MOVL C01710 V=800.0 PL=0
MOVL C01711 V=800.0 PL=0
MOVL C01712 V=800.0 PL=0
MOVL C01713 V=800.0 PL=0
MOVL C01714 V=800.0 PL=0
MOVL C01715 V=800.0 PL=0
MOVL C01716 V=800.0 PL=0
MOVL C01717 V=800.0 PL=0
MOVL C01718 V=800.0 PL=0
MOVL C01719 V=800.0 PL=0
MOVL C01720 V=800.0 PL=0
MOVL C01721 V=800.0 PL=0
MOVL C01722 V=800.0 PL=0
MOVL C01723 V=800.0 PL=0
MOVL C01724 V=800.0 PL=0
MOVL C01725 V=800.0 PL=0
MOVL C01726 V=800.0 PL=0
MOVL C01727 V=800.0 PL=0
MOVL C01728 V=800.0 PL=0
MOVL C01729 V=800.0 PL=0
MOVL C01730 V=800.0 PL=0
MOVL C01731 V=800.0 PL=0
MOVL C01732 V=800.0 PL=0
MOVL C01733 V=800.0 PL=0
MOVL C01734 V=800.0 PL=0
MOVL C01735 V=800.0 PL=0
MOVL C01736 V=800.0 PL=0
MOVL C01737 V=800.0 PL=0
MOVL C01738 V=800.0 PL=0
MOVL C01739 V=800.0 PL=0
MOVL C01740 V=800.0 PL=0
MOVL C01741 V=800.0 PL=0
MOVL C01742 V=800.0 PL=0
MOVL C01743 V=800.0 PL=0
MOVL C01744 V=800.0 PL=0
MOVL C01745 V=800.0 PL=0
MOVL C01746 V=800.0 PL=0
MOVL C01747 V=800.0 PL=0
MOVL C01748 V=800.0 PL=0
MOVL C01749 V=800.0 PL=0
MOVL C01750 V=800.0 PL=0
MOVL C01751 V=800.0 PL=0
MOVL C01752 V=800.0 PL=0
MOVL C01753 V=800.0 PL=0
MOVL C01754 V=800.0 PL=0
MOVL C01755 V=800.0 PL=0
MOVL C01756 V=800.0 PL=0
MOVL C01757 V=800.0 PL=0
MOVL C01758 V=800.0 PL=0
MOVL C01759 V=800.0 PL=0
MOVL C01760 V=800.0 PL=0
MOVL C01761 V=800.0 PL=0
MOVL C01762 V=800.0 PL=0
MOVL C01763 V=800.0 PL=0
MOVL C01764 V=800.0 PL=0
MOVL C01765 V=800.0 PL=0
MOVL C01766 V=800.0 PL=0
MOVL C01767 V=800.0 PL=0
MOVL C01768 V=800.0 PL=0
MOVL C01769 V=800.0 PL=0
MOVL C01770 V=800.0 PL=0
MOVL C01771 V=800.0 PL=0
MOVL C01772 V=800.0 PL=0
MOVL C01773 V=800.0 PL=0
MOVL C01774 V=800.0 PL=0
MOVL C01775 V=800.0 PL=0
MOVL C01776 V=800.0 PL=0
MOVL C01777 V=800.0 PL=0
MOVL C01778 V=800.0 PL=0
MOVL C01779 V=800.0 PL=0
MOVL C01780 V=800.0 PL=0
MOVL C01781 V=800.0 PL=0
MOVL C01782 V=800.0 PL=0
MOVL C01783 V=800.0 PL=0
MOVL C01784 V=800.0 PL=0
MOVL C01785 V=800.0 PL=0
MOVL C01786 V=800.0 PL=0
MOVL C01787 V=800.0 PL=0
MOVL C01788 V=800.0 PL=0
MOVL C01789 V=800.0 PL=0
MOVL C01790 V=800.0 PL=0
MOVL C01791 V=800.0 PL=0
MOVL C01792 V=800.0 PL=0
MOVL C01793 V=800.0 PL=0
MOVL C01794 V=800.0 PL=0
MOVL C01795 V=800.0 PL=0
MOVL C01796 V=800.0 PL=0
MOVL C01797 V=800.0 PL=0
MOVL C01798 V=800.0 PL=0
MOVL C01799 V=800.0 PL=0
MOVL C01800 V=800.0 PL=0
MOVL C01801 V=800.0 PL=0
MOVL C01802 V=800.0 PL=0
MOVL C01803 V=800.0 PL=0
